Yaskawa INFORM job: DEMO_ROOF_UPPER_0625_3PAINT_61.JBI

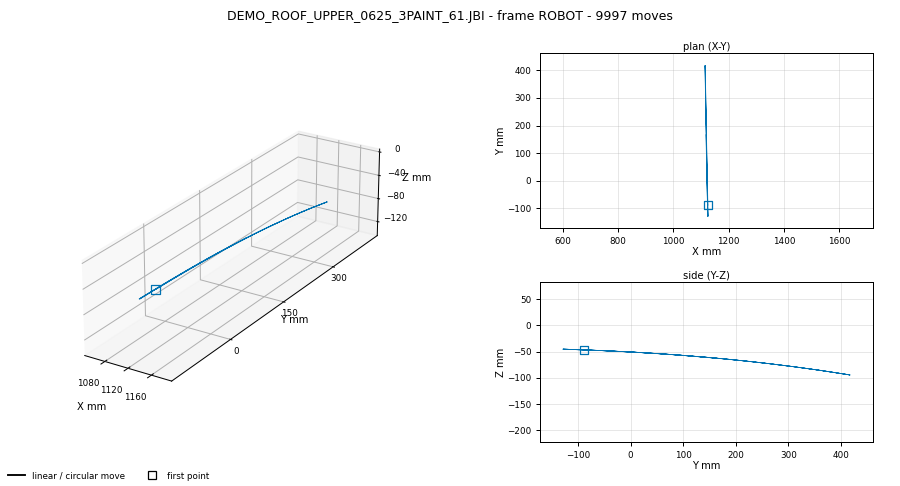
[picture p0: tool path of DEMO_ROOF_UPPER_0625_3PAINT_61.JBI in frame ROBOT, 9997 of 9997 moves have a stored position in this frame; points joined in program order, loops and branches not executed]
/JOB
//NAME DEMO_ROOF_UPPER_0625_3PAINT61
//POS
///NPOS 9997,0,0,0,0,0
///TOOL 0
///USER 0
///POSTYPE ROBOT
///RECTAN
///RCONF 1,0,0,0,0,0,0,0,0,0,0,0,0,0,0,0,0,0,0,0,0,0,0,0
C00000=1124.529,-88.514,-46.589,179.556,4.643,148.912
C00001=1124.524,-88.298,-46.597,179.556,4.647,148.913
C00002=1124.520,-88.083,-46.605,179.555,4.652,148.914
C00003=1124.516,-87.867,-46.613,179.555,4.656,148.915
C00004=1124.510,-87.651,-46.621,179.554,4.660,148.916
C00005=1124.505,-87.402,-46.630,179.554,4.665,148.917
C00006=1124.500,-87.152,-46.639,179.554,4.670,148.918
C00007=1124.494,-86.902,-46.649,179.553,4.675,148.920
C00008=1124.489,-86.652,-46.658,179.552,4.680,148.921
C00009=1124.484,-86.402,-46.667,179.552,4.685,148.922
C00010=1124.478,-86.152,-46.676,179.551,4.690,148.923
C00011=1124.473,-85.903,-46.686,179.551,4.695,148.925
C00012=1124.468,-85.653,-46.695,179.551,4.700,148.926
C00013=1124.462,-85.403,-46.704,179.551,4.705,148.927
C00014=1124.457,-85.154,-46.714,179.549,4.710,148.928
C00015=1124.452,-84.904,-46.723,179.549,4.715,148.929
C00016=1124.446,-84.654,-46.732,179.549,4.720,148.931
C00017=1124.441,-84.405,-46.742,179.549,4.725,148.932
C00018=1124.435,-84.154,-46.752,179.548,4.730,148.933
C00019=1124.430,-83.905,-46.760,179.548,4.735,148.934
C00020=1124.425,-83.655,-46.770,179.548,4.740,148.935
C00021=1124.419,-83.405,-46.780,179.548,4.745,148.936
C00022=1124.414,-83.155,-46.788,179.547,4.751,148.938
C00023=1124.409,-82.906,-46.799,179.547,4.756,148.939
C00024=1124.403,-82.656,-46.808,179.547,4.761,148.940
C00025=1124.398,-82.406,-46.817,179.546,4.766,148.941
C00026=1124.393,-82.157,-46.827,179.546,4.771,148.943
C00027=1124.388,-81.907,-46.836,179.546,4.776,148.944
C00028=1124.382,-81.657,-46.846,179.545,4.781,148.945
C00029=1124.377,-81.407,-46.855,179.545,4.786,148.946
C00030=1124.371,-81.157,-46.864,179.545,4.791,148.947
C00031=1124.366,-80.908,-46.874,179.545,4.796,148.948
C00032=1124.360,-80.658,-46.883,179.545,4.802,148.950
C00033=1124.356,-80.408,-46.893,179.545,4.807,148.951
C00034=1124.350,-80.158,-46.903,179.544,4.812,148.952
C00035=1124.345,-79.908,-46.912,179.544,4.817,148.953
C00036=1124.339,-79.658,-46.922,179.544,4.822,148.954
C00037=1124.334,-79.409,-46.931,179.544,4.827,148.955
C00038=1124.328,-79.159,-46.941,179.544,4.833,148.957
C00039=1124.324,-78.910,-46.951,179.544,4.838,148.958
C00040=1124.318,-78.659,-46.960,179.543,4.843,148.959
C00041=1124.313,-78.410,-46.970,179.543,4.848,148.960
C00042=1124.307,-78.160,-46.979,179.543,4.853,148.961
C00043=1124.302,-77.911,-46.989,179.543,4.858,148.962
C00044=1124.296,-77.661,-46.998,179.543,4.864,148.964
C00045=1124.291,-77.411,-47.008,179.543,4.870,148.965
C00046=1124.286,-77.161,-47.018,179.543,4.875,148.966
C00047=1124.280,-76.911,-47.028,179.543,4.879,148.967
C00048=1124.275,-76.662,-47.038,179.543,4.885,148.968
C00049=1124.270,-76.412,-47.047,179.543,4.890,148.969
C00050=1124.264,-76.162,-47.057,179.543,4.895,148.970
C00051=1124.259,-75.912,-47.066,179.543,4.901,148.972
C00052=1124.253,-75.663,-47.076,179.543,4.906,148.973
C00053=1124.249,-75.447,-47.084,179.543,4.910,148.974
C00054=1124.244,-75.231,-47.094,179.543,4.915,148.975
C00055=1124.240,-75.016,-47.101,179.544,4.920,148.975
C00056=1124.235,-74.800,-47.110,179.544,4.924,148.976
C00057=1124.231,-74.585,-47.118,179.544,4.928,148.977
C00058=1124.226,-74.369,-47.127,179.544,4.933,148.978
C00059=1124.222,-74.153,-47.135,179.543,4.937,148.979
C00060=1124.216,-73.938,-47.144,179.544,4.942,148.980
C00061=1124.212,-73.688,-47.153,179.544,4.947,148.981
C00062=1124.206,-73.438,-47.163,179.544,4.952,148.982
C00063=1124.201,-73.189,-47.174,179.545,4.958,148.984
C00064=1124.196,-72.939,-47.183,179.544,4.963,148.985
C00065=1124.190,-72.689,-47.193,179.545,4.968,148.986
C00066=1124.184,-72.440,-47.203,179.545,4.974,148.987
C00067=1124.179,-72.189,-47.214,179.545,4.979,148.988
C00068=1124.174,-71.940,-47.223,179.545,4.984,148.989
C00069=1124.168,-71.690,-47.233,179.546,4.990,148.990
C00070=1124.163,-71.441,-47.243,179.546,4.995,148.991
C00071=1124.158,-71.191,-47.252,179.546,5.000,148.992
C00072=1124.153,-70.941,-47.263,179.547,5.006,148.993
C00073=1124.147,-70.691,-47.273,179.547,5.010,148.994
C00074=1124.141,-70.441,-47.283,179.547,5.016,148.995
C00075=1124.137,-70.192,-47.292,179.548,5.021,148.996
C00076=1124.132,-69.942,-47.303,179.548,5.026,148.997
C00077=1124.126,-69.692,-47.313,179.549,5.032,148.998
C00078=1124.120,-69.443,-47.323,179.548,5.037,149.000
C00079=1124.116,-69.194,-47.333,179.549,5.043,149.000
C00080=1124.110,-68.943,-47.343,179.549,5.048,149.002
C00081=1124.105,-68.693,-47.353,179.550,5.053,149.003
C00082=1124.099,-68.444,-47.363,179.550,5.059,149.004
C00083=1124.094,-68.193,-47.374,179.550,5.063,149.005
C00084=1124.089,-67.944,-47.383,179.551,5.069,149.006
C00085=1124.084,-67.695,-47.394,179.551,5.074,149.007
C00086=1124.078,-67.445,-47.404,179.552,5.080,149.008
C00087=1124.073,-67.195,-47.414,179.552,5.085,149.009
C00088=1124.067,-66.945,-47.425,179.553,5.090,149.010
C00089=1124.062,-66.696,-47.435,179.554,5.095,149.011
C00090=1124.058,-66.446,-47.445,179.554,5.101,149.012
C00091=1124.052,-66.196,-47.455,179.554,5.106,149.013
C00092=1124.046,-65.947,-47.465,179.555,5.111,149.014
C00093=1124.041,-65.696,-47.476,179.555,5.117,149.015
C00094=1124.036,-65.447,-47.486,179.556,5.122,149.016
C00095=1124.030,-65.197,-47.496,179.557,5.128,149.017
C00096=1124.025,-64.947,-47.507,179.558,5.132,149.017
C00097=1124.020,-64.698,-47.517,179.559,5.138,149.018
C00098=1124.014,-64.448,-47.527,179.558,5.143,149.020
C00099=1124.010,-64.198,-47.537,179.559,5.149,149.020
C00100=1124.004,-63.949,-47.547,179.560,5.153,149.021
C00101=1123.998,-63.699,-47.558,179.561,5.159,149.022
C00102=1123.993,-63.449,-47.568,179.562,5.165,149.023
C00103=1123.988,-63.199,-47.578,179.562,5.169,149.024
C00104=1123.983,-62.950,-47.590,179.563,5.175,149.025
C00105=1123.978,-62.700,-47.600,179.564,5.180,149.026
C00106=1123.972,-62.451,-47.610,179.564,5.185,149.027
C00107=1123.967,-62.200,-47.621,179.565,5.191,149.028
C00108=1123.961,-61.951,-47.631,179.566,5.196,149.029
C00109=1123.957,-61.735,-47.640,179.567,5.201,149.030
C00110=1123.952,-61.520,-47.649,179.568,5.206,149.030
C00111=1123.948,-61.305,-47.658,179.568,5.210,149.031
C00112=1123.944,-61.089,-47.667,179.569,5.215,149.032
C00113=1123.939,-60.874,-47.677,179.570,5.219,149.033
C00114=1123.934,-60.658,-47.686,179.570,5.224,149.033
C00115=1123.929,-60.442,-47.695,179.571,5.228,149.034
C00116=1123.925,-60.226,-47.704,179.572,5.233,149.035
C00117=1123.920,-59.977,-47.715,179.571,5.237,149.036
C00118=1123.914,-59.727,-47.725,179.571,5.242,149.037
C00119=1123.909,-59.477,-47.736,179.571,5.246,149.038
C00120=1123.904,-59.228,-47.747,179.571,5.251,149.039
C00121=1123.898,-58.979,-47.757,179.571,5.256,149.040
C00122=1123.893,-58.728,-47.768,179.571,5.260,149.041
C00123=1123.888,-58.479,-47.778,179.571,5.265,149.042
C00124=1123.883,-58.229,-47.789,179.570,5.269,149.043
C00125=1123.878,-57.980,-47.799,179.570,5.274,149.045
C00126=1123.873,-57.729,-47.810,179.570,5.279,149.046
C00127=1123.867,-57.480,-47.821,179.570,5.284,149.047
C00128=1123.862,-57.230,-47.831,179.569,5.288,149.048
C00129=1123.856,-56.980,-47.842,179.569,5.293,149.049
C00130=1123.851,-56.731,-47.854,179.570,5.298,149.050
C00131=1123.846,-56.481,-47.864,179.569,5.302,149.051
C00132=1123.841,-56.232,-47.875,179.569,5.307,149.052
C00133=1123.836,-55.981,-47.886,179.569,5.311,149.053
C00134=1123.830,-55.732,-47.896,179.568,5.316,149.054
C00135=1123.826,-55.482,-47.907,179.568,5.320,149.055
C00136=1123.820,-55.233,-47.917,179.568,5.326,149.056
C00137=1123.815,-54.983,-47.929,179.568,5.331,149.057
C00138=1123.809,-54.733,-47.939,179.567,5.335,149.059
C00139=1123.804,-54.483,-47.950,179.568,5.340,149.059
C00140=1123.799,-54.234,-47.961,179.567,5.344,149.061
C00141=1123.794,-53.984,-47.972,179.567,5.349,149.062
C00142=1123.788,-53.735,-47.982,179.567,5.353,149.063
C00143=1123.783,-53.484,-47.994,179.567,5.358,149.064
C00144=1123.778,-53.235,-48.005,179.567,5.363,149.065
C00145=1123.772,-52.985,-48.015,179.567,5.367,149.066
C00146=1123.768,-52.735,-48.026,179.566,5.373,149.067
C00147=1123.762,-52.486,-48.037,179.566,5.377,149.068
C00148=1123.757,-52.236,-48.048,179.566,5.382,149.069
C00149=1123.751,-51.986,-48.059,179.565,5.386,149.070
C00150=1123.746,-51.737,-48.070,179.565,5.391,149.071
C00151=1123.741,-51.487,-48.081,179.566,5.396,149.072
C00152=1123.735,-51.237,-48.092,179.565,5.400,149.073
C00153=1123.730,-50.987,-48.103,179.565,5.405,149.075
C00154=1123.725,-50.738,-48.114,179.565,5.409,149.075
C00155=1123.720,-50.488,-48.124,179.565,5.415,149.077
C00156=1123.714,-50.239,-48.136,179.564,5.419,149.078
C00157=1123.709,-49.988,-48.146,179.564,5.424,149.079
C00158=1123.704,-49.739,-48.158,179.564,5.429,149.080
C00159=1123.698,-49.490,-48.169,179.564,5.433,149.081
C00160=1123.693,-49.239,-48.180,179.564,5.438,149.082
C00161=1123.689,-48.990,-48.191,179.564,5.442,149.083
C00162=1123.683,-48.740,-48.201,179.563,5.447,149.084
C00163=1123.678,-48.490,-48.213,179.563,5.452,149.085
C00164=1123.672,-48.241,-48.224,179.563,5.457,149.086
C00165=1123.668,-48.026,-48.233,179.563,5.461,149.087
C00166=1123.664,-47.810,-48.243,179.562,5.465,149.088
C00167=1123.659,-47.594,-48.252,179.562,5.469,149.089
C00168=1123.655,-47.379,-48.262,179.562,5.473,149.090
C00169=1123.650,-47.164,-48.271,179.562,5.477,149.091
C00170=1123.645,-46.948,-48.281,179.562,5.481,149.092
C00171=1123.641,-46.733,-48.291,179.562,5.485,149.093
C00172=1123.636,-46.518,-48.300,179.562,5.489,149.094
C00173=1123.631,-46.268,-48.312,179.561,5.494,149.095
C00174=1123.625,-46.018,-48.322,179.561,5.499,149.096
C00175=1123.620,-45.768,-48.334,179.562,5.503,149.097
C00176=1123.615,-45.519,-48.345,179.561,5.508,149.098
C00177=1123.610,-45.269,-48.356,179.561,5.513,149.099
C00178=1123.604,-45.019,-48.367,179.560,5.517,149.100
C00179=1123.600,-44.770,-48.379,179.561,5.522,149.101
C00180=1123.595,-44.520,-48.390,179.561,5.527,149.102
C00181=1123.589,-44.270,-48.401,179.560,5.532,149.104
C00182=1123.584,-44.021,-48.412,179.560,5.536,149.105
C00183=1123.578,-43.771,-48.424,179.560,5.541,149.106
C00184=1123.573,-43.521,-48.434,179.560,5.546,149.107
C00185=1123.568,-43.272,-48.445,179.559,5.550,149.108
C00186=1123.563,-43.022,-48.457,179.560,5.556,149.109
C00187=1123.557,-42.773,-48.468,179.562,5.561,149.109
C00188=1123.552,-42.523,-48.480,179.563,5.567,149.110
C00189=1123.547,-42.273,-48.491,179.565,5.572,149.111
C00190=1123.542,-42.023,-48.503,179.567,5.578,149.112
C00191=1123.536,-41.774,-48.514,179.568,5.584,149.113
C00192=1123.531,-41.524,-48.525,179.570,5.590,149.113
C00193=1123.526,-41.274,-48.537,179.572,5.595,149.114
C00194=1123.521,-41.024,-48.549,179.573,5.600,149.115
C00195=1123.515,-40.775,-48.560,179.574,5.606,149.115
C00196=1123.510,-40.525,-48.571,179.576,5.611,149.116
C00197=1123.505,-40.275,-48.582,179.577,5.617,149.117
C00198=1123.500,-40.025,-48.594,179.579,5.622,149.118
C00199=1123.494,-39.776,-48.605,179.580,5.627,149.118
C00200=1123.489,-39.526,-48.617,179.581,5.632,149.119
C00201=1123.484,-39.277,-48.628,179.582,5.637,149.120
C00202=1123.479,-39.027,-48.640,179.583,5.643,149.121
C00203=1123.473,-38.777,-48.652,179.585,5.648,149.122
C00204=1123.468,-38.528,-48.663,179.586,5.653,149.122
C00205=1123.463,-38.278,-48.675,179.587,5.658,149.123
C00206=1123.458,-38.028,-48.686,179.588,5.663,149.124
C00207=1123.452,-37.778,-48.698,179.589,5.668,149.125
C00208=1123.447,-37.528,-48.710,179.590,5.673,149.125
C00209=1123.442,-37.279,-48.721,179.591,5.678,149.126
C00210=1123.437,-37.029,-48.734,179.592,5.683,149.127
C00211=1123.432,-36.781,-48.744,179.593,5.688,149.128
C00212=1123.426,-36.531,-48.756,179.594,5.693,149.128
C00213=1123.421,-36.281,-48.768,179.595,5.698,149.129
C00214=1123.416,-36.031,-48.779,179.595,5.702,149.130
C00215=1123.411,-35.781,-48.791,179.596,5.707,149.131
C00216=1123.405,-35.531,-48.803,179.597,5.711,149.132
C00217=1123.400,-35.281,-48.815,179.598,5.716,149.133
C00218=1123.396,-35.032,-48.827,179.598,5.721,149.133
C00219=1123.390,-34.783,-48.839,179.598,5.725,149.134
C00220=1123.384,-34.533,-48.851,179.599,5.730,149.135
C00221=1123.380,-34.317,-48.861,179.600,5.734,149.136
C00222=1123.376,-34.103,-48.871,179.600,5.738,149.137
C00223=1123.371,-33.887,-48.881,179.601,5.741,149.137
C00224=1123.367,-33.671,-48.891,179.601,5.746,149.138
C00225=1123.362,-33.456,-48.902,179.601,5.750,149.139
C00226=1123.358,-33.241,-48.912,179.602,5.753,149.139
C00227=1123.353,-33.026,-48.922,179.602,5.757,149.140
C00228=1123.349,-32.810,-48.933,179.602,5.761,149.141
C00229=1123.344,-32.561,-48.944,179.602,5.766,149.142
C00230=1123.339,-32.311,-48.956,179.602,5.770,149.143
C00231=1123.333,-32.061,-48.968,179.603,5.774,149.144
C00232=1123.328,-31.812,-48.980,179.603,5.778,149.145
C00233=1123.322,-31.562,-48.992,179.603,5.783,149.146
C00234=1123.317,-31.313,-49.003,179.603,5.787,149.146
C00235=1123.312,-31.063,-49.015,179.603,5.791,149.147
C00236=1123.307,-30.813,-49.028,179.603,5.796,149.148
C00237=1123.301,-30.564,-49.040,179.603,5.800,149.149
C00238=1123.297,-30.314,-49.051,179.602,5.804,149.150
C00239=1123.292,-30.065,-49.064,179.602,5.808,149.151
C00240=1123.286,-29.815,-49.075,179.602,5.812,149.152
C00241=1123.281,-29.565,-49.087,179.602,5.817,149.153
C00242=1123.276,-29.315,-49.100,179.602,5.821,149.154
C00243=1123.270,-29.065,-49.112,179.601,5.825,149.155
C00244=1123.265,-28.816,-49.123,179.601,5.829,149.156
C00245=1123.260,-28.567,-49.136,179.600,5.833,149.157
C00246=1123.255,-28.317,-49.148,179.599,5.837,149.158
C00247=1123.250,-28.067,-49.160,179.599,5.841,149.159
C00248=1123.244,-27.817,-49.172,179.599,5.845,149.161
C00249=1123.239,-27.567,-49.184,179.598,5.850,149.162
C00250=1123.235,-27.318,-49.196,179.598,5.854,149.163
C00251=1123.229,-27.068,-49.208,179.597,5.857,149.164
C00252=1123.224,-26.819,-49.220,179.596,5.861,149.165
C00253=1123.219,-26.569,-49.232,179.595,5.866,149.166
C00254=1123.213,-26.319,-49.244,179.594,5.869,149.167
C00255=1123.208,-26.070,-49.257,179.594,5.874,149.168
C00256=1123.203,-25.820,-49.269,179.593,5.878,149.169
C00257=1123.198,-25.571,-49.281,179.593,5.883,149.170
C00258=1123.193,-25.321,-49.293,179.595,5.888,149.171
C00259=1123.188,-25.072,-49.305,179.595,5.893,149.172
C00260=1123.182,-24.822,-49.317,179.596,5.897,149.173
C00261=1123.177,-24.571,-49.329,179.597,5.903,149.174
C00262=1123.172,-24.322,-49.342,179.597,5.908,149.174
C00263=1123.167,-24.072,-49.354,179.598,5.912,149.175
C00264=1123.162,-23.823,-49.366,179.598,5.917,149.176
C00265=1123.156,-23.573,-49.378,179.599,5.923,149.177
C00266=1123.151,-23.323,-49.391,179.600,5.927,149.178
C00267=1123.146,-23.073,-49.403,179.601,5.932,149.179
C00268=1123.141,-22.824,-49.415,179.601,5.936,149.180
C00269=1123.135,-22.575,-49.428,179.602,5.942,149.181
C00270=1123.130,-22.325,-49.440,179.603,5.947,149.181
C00271=1123.125,-22.076,-49.452,179.603,5.951,149.182
C00272=1123.119,-21.826,-49.464,179.604,5.956,149.183
C00273=1123.114,-21.576,-49.477,179.605,5.961,149.184
C00274=1123.109,-21.326,-49.489,179.606,5.966,149.185
C00275=1123.104,-21.076,-49.502,179.606,5.971,149.186
C00276=1123.099,-20.827,-49.514,179.607,5.975,149.187
C00277=1123.095,-20.612,-49.524,179.608,5.980,149.187
C00278=1123.090,-20.396,-49.535,179.608,5.983,149.188
C00279=1123.085,-20.181,-49.546,179.609,5.988,149.189
C00280=1123.081,-19.967,-49.557,179.610,5.992,149.189
C00281=1123.077,-19.751,-49.568,179.610,5.996,149.190
C00282=1123.073,-19.536,-49.578,179.611,6.000,149.191
C00283=1123.068,-19.320,-49.589,179.611,6.004,149.191
C00284=1123.063,-19.106,-49.600,179.612,6.009,149.192
C00285=1123.058,-18.856,-49.612,179.613,6.013,149.193
C00286=1123.053,-18.606,-49.624,179.613,6.018,149.194
C00287=1123.048,-18.356,-49.637,179.614,6.022,149.195
C00288=1123.043,-18.106,-49.649,179.614,6.027,149.196
C00289=1123.038,-17.857,-49.662,179.616,6.032,149.196
C00290=1123.033,-17.608,-49.674,179.616,6.037,149.197
C00291=1123.027,-17.358,-49.687,179.617,6.042,149.198
C00292=1123.022,-17.108,-49.701,179.617,6.047,149.199
C00293=1123.017,-16.858,-49.712,179.618,6.051,149.200
C00294=1123.012,-16.609,-49.725,179.619,6.056,149.201
C00295=1123.006,-16.360,-49.738,179.619,6.060,149.201
C00296=1123.001,-16.110,-49.750,179.620,6.065,149.202
C00297=1122.997,-15.860,-49.763,179.621,6.069,149.203
C00298=1122.991,-15.610,-49.776,179.621,6.074,149.204
C00299=1122.986,-15.361,-49.788,179.622,6.079,149.205
C00300=1122.980,-15.111,-49.801,179.623,6.084,149.205
C00301=1122.975,-14.862,-49.814,179.624,6.089,149.206
C00302=1122.971,-14.612,-49.827,179.624,6.093,149.207
C00303=1122.966,-14.363,-49.839,179.625,6.098,149.208
C00304=1122.960,-14.113,-49.852,179.626,6.103,149.209
C00305=1122.954,-13.863,-49.864,179.626,6.107,149.210
C00306=1122.950,-13.613,-49.877,179.627,6.112,149.210
C00307=1122.945,-13.364,-49.890,179.628,6.116,149.211
C00308=1122.939,-13.114,-49.903,179.628,6.121,149.212
C00309=1122.934,-12.864,-49.916,179.629,6.126,149.213
C00310=1122.929,-12.615,-49.929,179.630,6.130,149.214
C00311=1122.924,-12.365,-49.941,179.630,6.135,149.215
C00312=1122.918,-12.116,-49.954,179.631,6.140,149.215
C00313=1122.914,-11.866,-49.967,179.632,6.144,149.216
C00314=1122.909,-11.617,-49.980,179.632,6.149,149.217
C00315=1122.903,-11.367,-49.992,179.633,6.153,149.218
C00316=1122.898,-11.117,-50.006,179.634,6.158,149.219
C00317=1122.893,-10.868,-50.019,179.634,6.162,149.219
C00318=1122.888,-10.618,-50.031,179.635,6.167,149.220
C00319=1122.882,-10.369,-50.044,179.636,6.172,149.221
C00320=1122.878,-10.119,-50.057,179.636,6.176,149.222
C00321=1122.872,-9.869,-50.070,179.637,6.181,149.223
C00322=1122.867,-9.620,-50.083,179.638,6.185,149.223
C00323=1122.862,-9.370,-50.096,179.638,6.190,149.224
C00324=1122.857,-9.121,-50.109,179.639,6.195,149.225
C00325=1122.853,-8.871,-50.122,179.640,6.199,149.226
C00326=1122.847,-8.621,-50.136,179.640,6.204,149.227
C00327=1122.842,-8.372,-50.148,179.641,6.209,149.228
C00328=1122.836,-8.122,-50.162,179.642,6.213,149.228
C00329=1122.831,-7.872,-50.174,179.642,6.218,149.229
C00330=1122.826,-7.623,-50.187,179.643,6.222,149.230
C00331=1122.821,-7.373,-50.201,179.644,6.227,149.231
C00332=1122.816,-7.124,-50.214,179.644,6.231,149.232
C00333=1122.812,-6.908,-50.225,179.645,6.235,149.232
C00334=1122.807,-6.694,-50.236,179.645,6.239,149.233
C00335=1122.803,-6.478,-50.248,179.646,6.243,149.234
C00336=1122.799,-6.263,-50.260,179.646,6.247,149.234
C00337=1122.793,-6.048,-50.270,179.646,6.250,149.235
C00338=1122.789,-5.833,-50.282,179.647,6.255,149.236
C00339=1122.785,-5.618,-50.293,179.648,6.258,149.236
C00340=1122.780,-5.403,-50.305,179.649,6.263,149.237
C00341=1122.775,-5.153,-50.317,179.649,6.267,149.238
C00342=1122.770,-4.903,-50.331,179.649,6.271,149.239
C00343=1122.765,-4.654,-50.344,179.650,6.276,149.240
C00344=1122.760,-4.404,-50.358,179.651,6.280,149.240
C00345=1122.755,-4.155,-50.370,179.651,6.285,149.241
C00346=1122.750,-3.905,-50.383,179.652,6.290,149.242
C00347=1122.744,-3.655,-50.397,179.653,6.294,149.243
C00348=1122.740,-3.406,-50.410,179.653,6.299,149.244
C00349=1122.734,-3.156,-50.424,179.654,6.304,149.245
C00350=1122.729,-2.907,-50.436,179.655,6.308,149.245
C00351=1122.724,-2.657,-50.450,179.655,6.312,149.246
C00352=1122.718,-2.407,-50.464,179.655,6.317,149.247
C00353=1122.714,-2.157,-50.477,179.656,6.321,149.248
C00354=1122.708,-1.908,-50.490,179.657,6.326,149.249
C00355=1122.704,-1.658,-50.503,179.657,6.330,149.250
C00356=1122.698,-1.409,-50.517,179.658,6.335,149.250
C00357=1122.694,-1.159,-50.530,179.659,6.339,149.251
C00358=1122.688,-0.910,-50.544,179.659,6.343,149.252
C00359=1122.684,-0.660,-50.557,179.659,6.348,149.253
C00360=1122.678,-0.411,-50.570,179.660,6.353,149.254
C00361=1122.673,-0.161,-50.585,179.661,6.357,149.254
C00362=1122.668,0.088,-50.597,179.661,6.362,149.255
C00363=1122.662,0.339,-50.611,179.662,6.367,149.256
C00364=1122.658,0.587,-50.624,179.662,6.371,149.257
C00365=1122.652,0.838,-50.638,179.663,6.375,149.258
C00366=1122.647,1.087,-50.652,179.663,6.379,149.259
C00367=1122.642,1.337,-50.665,179.664,6.384,149.259
C00368=1122.637,1.586,-50.678,179.664,6.389,149.260
C00369=1122.632,1.836,-50.691,179.665,6.393,149.261
C00370=1122.627,2.085,-50.705,179.666,6.398,149.262
C00371=1122.621,2.335,-50.719,179.666,6.403,149.263
C00372=1122.617,2.584,-50.732,179.666,6.407,149.264
C00373=1122.611,2.834,-50.746,179.667,6.411,149.265
C00374=1122.606,3.083,-50.760,179.668,6.416,149.265
C00375=1122.601,3.333,-50.773,179.668,6.420,149.266
C00376=1122.596,3.583,-50.787,179.669,6.425,149.267
C00377=1122.591,3.832,-50.801,179.669,6.429,149.268
C00378=1122.586,4.082,-50.814,179.669,6.434,149.269
C00379=1122.581,4.331,-50.828,179.670,6.438,149.269
C00380=1122.575,4.581,-50.841,179.671,6.443,149.270
C00381=1122.570,4.831,-50.856,179.672,6.448,149.271
C00382=1122.566,5.080,-50.869,179.672,6.452,149.272
C00383=1122.560,5.330,-50.882,179.672,6.456,149.273
C00384=1122.555,5.579,-50.896,179.673,6.461,149.274
C00385=1122.550,5.829,-50.911,179.673,6.466,149.275
C00386=1122.545,6.079,-50.924,179.674,6.470,149.275
C00387=1122.540,6.328,-50.938,179.675,6.475,149.276
C00388=1122.535,6.577,-50.952,179.675,6.479,149.277
C00389=1122.531,6.793,-50.963,179.675,6.483,149.278
C00390=1122.526,7.007,-50.975,179.676,6.487,149.279
C00391=1122.522,7.223,-50.986,179.676,6.490,149.279
C00392=1122.517,7.438,-50.999,179.676,6.495,149.280
C00393=1122.513,7.653,-51.011,179.677,6.499,149.281
C00394=1122.508,7.867,-51.022,179.677,6.502,149.282
C00395=1122.504,8.083,-51.034,179.677,6.506,149.282
C00396=1122.499,8.298,-51.046,179.678,6.510,149.283
C00397=1122.495,8.548,-51.060,179.679,6.515,149.284
C00398=1122.489,8.797,-51.074,179.679,6.520,149.285
C00399=1122.484,9.046,-51.088,179.680,6.524,149.285
C00400=1122.479,9.297,-51.102,179.681,6.529,149.286
C00401=1122.473,9.546,-51.116,179.681,6.534,149.287
C00402=1122.469,9.795,-51.130,179.682,6.538,149.288
C00403=1122.464,10.045,-51.144,179.683,6.543,149.289
C00404=1122.459,10.294,-51.158,179.684,6.548,149.290
C00405=1122.453,10.544,-51.171,179.685,6.552,149.290
C00406=1122.449,10.794,-51.185,179.686,6.557,149.291
C00407=1122.443,11.043,-51.199,179.686,6.562,149.292
C00408=1122.438,11.292,-51.214,179.687,6.566,149.293
C00409=1122.433,11.542,-51.228,179.688,6.571,149.294
C00410=1122.428,11.792,-51.242,179.689,6.575,149.294
C00411=1122.423,12.041,-51.256,179.689,6.580,149.295
C00412=1122.418,12.290,-51.270,179.690,6.585,149.296
C00413=1122.413,12.541,-51.283,179.691,6.589,149.297
C00414=1122.408,12.790,-51.298,179.692,6.594,149.298
C00415=1122.403,13.039,-51.312,179.693,6.599,149.298
C00416=1122.398,13.289,-51.326,179.694,6.604,149.299
C00417=1122.393,13.539,-51.340,179.695,6.608,149.300
C00418=1122.388,13.788,-51.354,179.695,6.613,149.301
C00419=1122.382,14.037,-51.368,179.696,6.617,149.301
C00420=1122.377,14.287,-51.383,179.697,6.622,149.302
C00421=1122.372,14.537,-51.397,179.698,6.626,149.303
C00422=1122.367,14.787,-51.411,179.699,6.631,149.304
C00423=1122.362,15.036,-51.425,179.699,6.635,149.305
C00424=1122.357,15.285,-51.439,179.700,6.640,149.305
C00425=1122.352,15.535,-51.454,179.701,6.644,149.306
C00426=1122.347,15.785,-51.468,179.702,6.649,149.307
C00427=1122.342,16.034,-51.482,179.703,6.653,149.307
C00428=1122.336,16.283,-51.496,179.703,6.658,149.308
C00429=1122.331,16.533,-51.510,179.705,6.663,149.309
C00430=1122.326,16.783,-51.525,179.706,6.668,149.310
C00431=1122.322,17.032,-51.540,179.707,6.672,149.310
C00432=1122.317,17.282,-51.554,179.707,6.677,149.311
C00433=1122.311,17.531,-51.568,179.708,6.681,149.312
C00434=1122.306,17.780,-51.582,179.709,6.685,149.313
C00435=1122.301,18.030,-51.596,179.710,6.690,149.313
C00436=1122.296,18.280,-51.611,179.711,6.694,149.314
C00437=1122.291,18.530,-51.626,179.711,6.699,149.315
C00438=1122.286,18.779,-51.641,179.712,6.703,149.316
C00439=1122.281,19.028,-51.654,179.713,6.708,149.316
C00440=1122.276,19.278,-51.669,179.714,6.712,149.317
C00441=1122.271,19.527,-51.683,179.715,6.717,149.318
C00442=1122.266,19.777,-51.697,179.716,6.721,149.318
C00443=1122.261,20.026,-51.712,179.717,6.726,149.319
C00444=1122.256,20.276,-51.727,179.718,6.730,149.320
C00445=1122.251,20.491,-51.739,179.719,6.734,149.321
C00446=1122.247,20.706,-51.752,179.719,6.738,149.321
C00447=1122.243,20.921,-51.764,179.720,6.742,149.322
C00448=1122.238,21.136,-51.777,179.721,6.745,149.322
C00449=1122.234,21.351,-51.789,179.722,6.750,149.323
C00450=1122.229,21.566,-51.802,179.723,6.753,149.324
C00451=1122.225,21.781,-51.814,179.724,6.758,149.324
C00452=1122.221,21.996,-51.827,179.724,6.761,149.325
C00453=1122.215,22.245,-51.841,179.725,6.765,149.326
C00454=1122.210,22.495,-51.855,179.726,6.770,149.326
C00455=1122.206,22.744,-51.870,179.727,6.774,149.327
C00456=1122.200,22.994,-51.885,179.728,6.779,149.328
C00457=1122.195,23.243,-51.900,179.729,6.783,149.328
C00458=1122.190,23.492,-51.915,179.730,6.787,149.329
C00459=1122.185,23.742,-51.929,179.731,6.792,149.330
C00460=1122.180,23.992,-51.944,179.732,6.796,149.331
C00461=1122.175,24.241,-51.959,179.733,6.801,149.331
C00462=1122.170,24.491,-51.973,179.734,6.805,149.332
C00463=1122.165,24.740,-51.988,179.735,6.809,149.333
C00464=1122.160,24.990,-52.003,179.736,6.814,149.333
C00465=1122.155,25.240,-52.017,179.737,6.818,149.334
C00466=1122.150,25.489,-52.032,179.737,6.823,149.335
C00467=1122.144,25.739,-52.047,179.738,6.827,149.335
C00468=1122.140,25.988,-52.062,179.739,6.831,149.336
C00469=1122.135,26.238,-52.076,179.741,6.836,149.337
C00470=1122.130,26.487,-52.092,179.742,6.840,149.337
C00471=1122.125,26.737,-52.106,179.743,6.844,149.338
C00472=1122.120,26.986,-52.121,179.744,6.849,149.339
C00473=1122.114,27.236,-52.136,179.744,6.853,149.340
C00474=1122.110,27.485,-52.151,179.745,6.858,149.340
C00475=1122.105,27.735,-52.165,179.746,6.862,149.341
C00476=1122.099,27.984,-52.181,179.747,6.866,149.342
C00477=1122.094,28.234,-52.195,179.748,6.871,149.342
C00478=1122.090,28.483,-52.210,179.750,6.875,149.343
C00479=1122.084,28.732,-52.226,179.751,6.879,149.343
C00480=1122.079,28.982,-52.240,179.752,6.883,149.344
C00481=1122.074,29.231,-52.256,179.753,6.888,149.345
C00482=1122.069,29.481,-52.270,179.754,6.892,149.345
C00483=1122.064,29.730,-52.285,179.755,6.896,149.346
C00484=1122.059,29.980,-52.300,179.756,6.901,149.347
C00485=1122.054,30.229,-52.315,179.757,6.905,149.347
C00486=1122.049,30.479,-52.330,179.758,6.909,149.348
C00487=1122.044,30.728,-52.345,179.759,6.914,149.349
C00488=1122.039,30.979,-52.361,179.760,6.918,149.349
C00489=1122.034,31.228,-52.376,179.761,6.922,149.350
C00490=1122.030,31.477,-52.391,179.762,6.927,149.351
C00491=1122.024,31.727,-52.405,179.763,6.931,149.351
C00492=1122.019,31.976,-52.420,179.764,6.935,149.352
C00493=1122.014,32.225,-52.436,179.765,6.940,149.353
C00494=1122.009,32.475,-52.450,179.766,6.944,149.353
C00495=1122.003,32.724,-52.466,179.768,6.948,149.354
C00496=1121.999,32.974,-52.481,179.769,6.952,149.355
C00497=1121.994,33.224,-52.497,179.770,6.957,149.355
C00498=1121.989,33.473,-52.511,179.771,6.961,149.356
C00499=1121.984,33.723,-52.527,179.772,6.965,149.356
C00500=1121.978,33.972,-52.542,179.772,6.969,149.357
C00501=1121.974,34.187,-52.555,179.774,6.973,149.358
C00502=1121.970,34.401,-52.568,179.774,6.976,149.358
C00503=1121.966,34.616,-52.581,179.776,6.980,149.359
C00504=1121.962,34.832,-52.595,179.776,6.984,149.359
C00505=1121.957,35.047,-52.608,179.778,6.988,149.360
C00506=1121.953,35.261,-52.621,179.778,6.991,149.360
C00507=1121.948,35.476,-52.634,179.779,6.994,149.361
C00508=1121.944,35.691,-52.647,179.780,6.999,149.361
C00509=1121.939,35.940,-52.662,179.781,7.003,149.362
C00510=1121.934,36.190,-52.678,179.782,7.007,149.363
C00511=1121.929,36.439,-52.693,179.783,7.012,149.363
C00512=1121.924,36.689,-52.709,179.785,7.016,149.364
C00513=1121.919,36.938,-52.724,179.786,7.020,149.364
C00514=1121.914,37.187,-52.739,179.786,7.023,149.365
C00515=1121.908,37.437,-52.754,179.787,7.028,149.366
C00516=1121.904,37.687,-52.770,179.789,7.032,149.366
C00517=1121.899,37.936,-52.785,179.790,7.036,149.367
C00518=1121.893,38.186,-52.801,179.791,7.040,149.368
C00519=1121.889,38.435,-52.816,179.792,7.045,149.368
C00520=1121.884,38.685,-52.832,179.793,7.049,149.369
C00521=1121.879,38.934,-52.847,179.794,7.053,149.369
C00522=1121.873,39.184,-52.863,179.795,7.057,149.370
C00523=1121.869,39.433,-52.878,179.797,7.061,149.371
C00524=1121.864,39.683,-52.894,179.798,7.066,149.371
C00525=1121.858,39.932,-52.910,179.799,7.070,149.372
C00526=1121.854,40.181,-52.925,179.800,7.074,149.372
C00527=1121.849,40.430,-52.941,179.801,7.079,149.373
C00528=1121.844,40.680,-52.957,179.803,7.083,149.374
C00529=1121.838,40.930,-52.972,179.804,7.087,149.374
C00530=1121.834,41.179,-52.987,179.805,7.091,149.375
C00531=1121.828,41.428,-53.003,179.806,7.095,149.375
C00532=1121.824,41.678,-53.019,179.807,7.099,149.376
C00533=1121.818,41.928,-53.035,179.808,7.103,149.377
C00534=1121.814,42.177,-53.050,179.809,7.107,149.377
C00535=1121.809,42.427,-53.065,179.810,7.112,149.378
C00536=1121.804,42.676,-53.082,179.812,7.115,149.378
C00537=1121.798,42.925,-53.097,179.813,7.120,149.379
C00538=1121.794,43.175,-53.113,179.814,7.124,149.380
C00539=1121.789,43.424,-53.128,179.815,7.128,149.380
C00540=1121.784,43.674,-53.144,179.817,7.132,149.381
C00541=1121.779,43.923,-53.161,179.818,7.137,149.381
C00542=1121.774,44.173,-53.176,179.819,7.141,149.382
C00543=1121.768,44.422,-53.192,179.820,7.145,149.382
C00544=1121.763,44.672,-53.208,179.821,7.149,149.383
C00545=1121.759,44.921,-53.223,179.822,7.153,149.384
C00546=1121.754,45.170,-53.239,179.824,7.157,149.384
C00547=1121.749,45.420,-53.255,179.824,7.161,149.385
C00548=1121.744,45.669,-53.271,179.825,7.165,149.385
C00549=1121.739,45.918,-53.287,179.827,7.169,149.386
C00550=1121.734,46.168,-53.303,179.828,7.173,149.386
C00551=1121.728,46.418,-53.318,179.830,7.177,149.387
C00552=1121.724,46.667,-53.335,179.831,7.182,149.388
C00553=1121.719,46.916,-53.350,179.832,7.186,149.388
C00554=1121.714,47.166,-53.366,179.833,7.190,149.389
C00555=1121.709,47.415,-53.382,179.834,7.194,149.389
C00556=1121.704,47.665,-53.398,179.836,7.198,149.390
C00557=1121.700,47.880,-53.412,179.836,7.202,149.390
C00558=1121.695,48.095,-53.426,179.838,7.205,149.391
C00559=1121.691,48.309,-53.439,179.839,7.209,149.391
C00560=1121.687,48.524,-53.453,179.839,7.212,149.392
C00561=1121.683,48.739,-53.467,179.841,7.216,149.392
C00562=1121.678,48.953,-53.481,179.842,7.219,149.393
C00563=1121.674,49.169,-53.494,179.843,7.223,149.393
C00564=1121.669,49.383,-53.508,179.844,7.227,149.394
C00565=1121.664,49.632,-53.525,179.845,7.231,149.394
C00566=1121.659,49.882,-53.541,179.847,7.235,149.395
C00567=1121.654,50.131,-53.557,179.848,7.239,149.395
C00568=1121.650,50.381,-53.573,179.849,7.243,149.396
C00569=1121.644,50.630,-53.589,179.851,7.247,149.396
C00570=1121.640,50.880,-53.605,179.851,7.250,149.397
C00571=1121.635,51.129,-53.621,179.853,7.254,149.397
C00572=1121.630,51.379,-53.637,179.854,7.259,149.398
C00573=1121.625,51.628,-53.654,179.855,7.263,149.399
C00574=1121.620,51.878,-53.670,179.856,7.267,149.399
C00575=1121.615,52.126,-53.686,179.858,7.271,149.400
C00576=1121.610,52.377,-53.702,179.859,7.275,149.400
C00577=1121.605,52.625,-53.718,179.860,7.279,149.401
C00578=1121.601,52.875,-53.735,179.862,7.283,149.401
C00579=1121.595,53.124,-53.750,179.863,7.288,149.402
C00580=1121.591,53.374,-53.767,179.864,7.292,149.402
C00581=1121.585,53.623,-53.783,179.865,7.296,149.403
C00582=1121.580,53.873,-53.800,179.867,7.300,149.404
C00583=1121.575,54.122,-53.816,179.868,7.303,149.404
C00584=1121.570,54.372,-53.832,179.869,7.307,149.405
C00585=1121.565,54.621,-53.849,179.870,7.311,149.405
C00586=1121.561,54.870,-53.865,179.872,7.315,149.406
C00587=1121.555,55.119,-53.881,179.873,7.320,149.406
C00588=1121.550,55.369,-53.898,179.874,7.324,149.407
C00589=1121.546,55.619,-53.915,179.875,7.328,149.407
C00590=1121.540,55.868,-53.930,179.877,7.332,149.408
C00591=1121.536,56.118,-53.947,179.878,7.336,149.408
C00592=1121.531,56.366,-53.963,179.880,7.340,149.409
C00593=1121.526,56.616,-53.980,179.881,7.344,149.410
C00594=1121.520,56.866,-53.996,179.882,7.348,149.410
C00595=1121.516,57.115,-54.013,179.883,7.351,149.410
C00596=1121.511,57.365,-54.030,179.884,7.356,149.411
C00597=1121.506,57.613,-54.046,179.886,7.360,149.411
C00598=1121.501,57.863,-54.063,179.887,7.364,149.412
C00599=1121.495,58.113,-54.079,179.889,7.368,149.413
C00600=1121.491,58.362,-54.095,179.890,7.372,149.413
C00601=1121.486,58.612,-54.112,179.891,7.376,149.414
C00602=1121.481,58.861,-54.129,179.892,7.380,149.414
C00603=1121.476,59.110,-54.146,179.894,7.384,149.415
C00604=1121.472,59.360,-54.162,179.895,7.388,149.415
C00605=1121.466,59.609,-54.178,179.897,7.392,149.416
C00606=1121.461,59.859,-54.195,179.898,7.396,149.416
C00607=1121.457,60.108,-54.212,179.899,7.401,149.417
C00608=1121.451,60.357,-54.228,179.900,7.404,149.417
C00609=1121.446,60.607,-54.245,179.902,7.408,149.418
C00610=1121.442,60.856,-54.262,179.903,7.412,149.418
C00611=1121.437,61.105,-54.278,179.904,7.416,149.419
C00612=1121.431,61.355,-54.296,179.906,7.420,149.419
C00613=1121.427,61.569,-54.309,179.907,7.424,149.420
C00614=1121.423,61.785,-54.324,179.908,7.427,149.420
C00615=1121.419,61.998,-54.338,179.909,7.430,149.421
C00616=1121.414,62.214,-54.353,179.911,7.434,149.421
C00617=1121.411,62.429,-54.367,179.911,7.437,149.422
C00618=1121.406,62.643,-54.382,179.912,7.440,149.422
C00619=1121.402,62.858,-54.396,179.914,7.444,149.422
C00620=1121.397,63.072,-54.411,179.915,7.447,149.423
C00621=1121.393,63.321,-54.428,179.916,7.451,149.423
C00622=1121.388,63.571,-54.445,179.918,7.456,149.424
C00623=1121.383,63.820,-54.461,179.919,7.460,149.424
C00624=1121.378,64.069,-54.478,179.921,7.463,149.425
C00625=1121.373,64.319,-54.495,179.922,7.468,149.425
C00626=1121.368,64.569,-54.512,179.923,7.472,149.426
C00627=1121.363,64.818,-54.529,179.925,7.476,149.426
C00628=1121.358,65.067,-54.546,179.926,7.480,149.427
C00629=1121.353,65.317,-54.563,179.928,7.484,149.427
C00630=1121.348,65.566,-54.580,179.928,7.487,149.428
C00631=1121.343,65.815,-54.596,179.930,7.491,149.428
C00632=1121.339,66.064,-54.614,179.931,7.495,149.429
C00633=1121.334,66.314,-54.631,179.932,7.499,149.430
C00634=1121.329,66.564,-54.648,179.934,7.503,149.430
C00635=1121.324,66.813,-54.664,179.936,7.507,149.430
C00636=1121.319,67.062,-54.681,179.937,7.511,149.431
C00637=1121.314,67.311,-54.699,179.938,7.515,149.431
C00638=1121.309,67.561,-54.716,179.940,7.519,149.432
C00639=1121.305,67.810,-54.733,179.941,7.523,149.432
C00640=1121.299,68.060,-54.750,179.942,7.527,149.433
C00641=1121.294,68.309,-54.768,179.944,7.531,149.433
C00642=1121.289,68.558,-54.784,179.946,7.535,149.434
C00643=1121.284,68.808,-54.801,179.947,7.540,149.434
C00644=1121.280,69.057,-54.818,179.948,7.543,149.435
C00645=1121.275,69.307,-54.836,179.949,7.547,149.435
C00646=1121.270,69.555,-54.852,179.950,7.551,149.436
C00647=1121.265,69.805,-54.870,179.952,7.555,149.436
C00648=1121.260,70.054,-54.888,179.953,7.559,149.437
C00649=1121.255,70.304,-54.904,179.955,7.563,149.437
C00650=1121.250,70.554,-54.922,179.956,7.567,149.438
C00651=1121.246,70.802,-54.939,179.958,7.571,149.438
C00652=1121.241,71.052,-54.956,179.959,7.575,149.439
C00653=1121.235,71.301,-54.973,179.960,7.579,149.439
C00654=1121.231,71.550,-54.991,179.962,7.583,149.440
C00655=1121.225,71.800,-55.008,179.964,7.587,149.440
C00656=1121.220,72.049,-55.026,179.965,7.591,149.441
C00657=1121.216,72.299,-55.042,179.966,7.595,149.441
C00658=1121.211,72.548,-55.060,179.968,7.599,149.442
C00659=1121.206,72.798,-55.078,179.969,7.603,149.442
C00660=1121.201,73.047,-55.094,179.971,7.607,149.443
C00661=1121.196,73.296,-55.112,179.972,7.611,149.443
C00662=1121.191,73.546,-55.130,179.973,7.614,149.444
C00663=1121.186,73.794,-55.147,179.975,7.618,149.444
C00664=1121.181,74.044,-55.164,179.976,7.622,149.445
C00665=1121.176,74.293,-55.182,179.977,7.626,149.445
C00666=1121.171,74.543,-55.199,179.979,7.630,149.446
C00667=1121.167,74.792,-55.217,179.981,7.634,149.446
C00668=1121.162,75.041,-55.235,179.982,7.638,149.447
C00669=1121.158,75.256,-55.249,179.983,7.642,149.447
C00670=1121.153,75.471,-55.265,179.985,7.645,149.447
C00671=1121.149,75.685,-55.280,179.986,7.648,149.448
C00672=1121.145,75.900,-55.294,179.987,7.652,149.448
C00673=1121.141,76.114,-55.310,179.988,7.655,149.449
C00674=1121.137,76.329,-55.325,179.990,7.659,149.449
C00675=1121.132,76.543,-55.340,179.991,7.662,149.450
C00676=1121.128,76.758,-55.355,179.992,7.665,149.450
C00677=1121.123,77.008,-55.373,179.993,7.669,149.451
C00678=1121.118,77.257,-55.391,179.994,7.673,149.451
C00679=1121.114,77.506,-55.407,179.995,7.677,149.452
C00680=1121.109,77.755,-55.425,179.996,7.680,149.452
C00681=1121.104,78.005,-55.443,179.997,7.684,149.453
C00682=1121.099,78.254,-55.461,179.997,7.688,149.453
C00683=1121.094,78.504,-55.479,179.999,7.692,149.454
C00684=1121.089,78.753,-55.497,180.000,7.695,149.454
C00685=1121.084,79.002,-55.513,-179.999,7.699,149.455
C00686=1121.079,79.251,-55.531,-179.998,7.702,149.456
C00687=1121.074,79.501,-55.549,-179.997,7.706,149.456
C00688=1121.069,79.750,-55.567,-179.996,7.710,149.457
C00689=1121.064,80.000,-55.585,-179.995,7.714,149.457
C00690=1121.059,80.249,-55.602,-179.994,7.717,149.458
C00691=1121.054,80.498,-55.620,-179.993,7.721,149.458
C00692=1121.050,80.747,-55.638,-179.992,7.725,149.459
C00693=1121.045,80.996,-55.656,-179.991,7.729,149.459
C00694=1121.040,81.246,-55.673,-179.990,7.732,149.460
C00695=1121.036,81.496,-55.691,-179.988,7.736,149.460
C00696=1121.031,81.745,-55.709,-179.987,7.740,149.461
C00697=1121.026,81.994,-55.727,-179.986,7.743,149.461
C00698=1121.021,82.243,-55.745,-179.985,7.748,149.462
C00699=1121.016,82.493,-55.763,-179.984,7.751,149.462
C00700=1121.011,82.742,-55.781,-179.983,7.755,149.463
C00701=1121.006,82.991,-55.799,-179.982,7.759,149.463
C00702=1121.001,83.240,-55.817,-179.981,7.762,149.464
C00703=1120.996,83.490,-55.835,-179.979,7.766,149.465
C00704=1120.991,83.739,-55.853,-179.978,7.770,149.465
C00705=1120.986,83.988,-55.871,-179.977,7.774,149.466
C00706=1120.982,84.238,-55.889,-179.976,7.778,149.466
C00707=1120.977,84.487,-55.907,-179.975,7.782,149.467
C00708=1120.972,84.737,-55.924,-179.974,7.785,149.467
C00709=1120.967,84.986,-55.942,-179.972,7.789,149.468
C00710=1120.962,85.235,-55.960,-179.971,7.793,149.468
C00711=1120.957,85.484,-55.978,-179.969,7.797,149.469
C00712=1120.952,85.734,-55.996,-179.968,7.800,149.469
C00713=1120.947,85.983,-56.014,-179.967,7.804,149.470
C00714=1120.943,86.233,-56.032,-179.966,7.808,149.470
C00715=1120.938,86.482,-56.050,-179.965,7.811,149.471
C00716=1120.933,86.731,-56.068,-179.964,7.816,149.471
C00717=1120.928,86.980,-56.086,-179.962,7.820,149.472
C00718=1120.923,87.229,-56.104,-179.960,7.824,149.472
C00719=1120.918,87.479,-56.123,-179.959,7.828,149.473
C00720=1120.913,87.729,-56.141,-179.958,7.831,149.473
C00721=1120.909,87.977,-56.160,-179.957,7.835,149.474
C00722=1120.904,88.226,-56.178,-179.956,7.839,149.474
C00723=1120.899,88.476,-56.196,-179.954,7.843,149.475
C00724=1120.894,88.725,-56.214,-179.952,7.847,149.475
C00725=1120.890,88.939,-56.229,-179.951,7.850,149.476
C00726=1120.886,89.154,-56.245,-179.950,7.853,149.476
C00727=1120.881,89.369,-56.261,-179.949,7.857,149.476
C00728=1120.877,89.583,-56.277,-179.948,7.860,149.477
C00729=1120.873,89.797,-56.293,-179.947,7.863,149.477
C00730=1120.869,90.012,-56.308,-179.945,7.867,149.477
C00731=1120.865,90.227,-56.324,-179.944,7.870,149.478
C00732=1120.861,90.441,-56.340,-179.943,7.873,149.478
C00733=1120.856,90.690,-56.358,-179.941,7.877,149.479
C00734=1120.851,90.940,-56.376,-179.940,7.881,149.479
C00735=1120.846,91.189,-56.394,-179.939,7.885,149.480
C00736=1120.842,91.439,-56.413,-179.937,7.889,149.480
C00737=1120.837,91.687,-56.431,-179.935,7.893,149.481
C00738=1120.831,91.937,-56.450,-179.934,7.897,149.481
C00739=1120.826,92.186,-56.468,-179.932,7.901,149.482
C00740=1120.822,92.436,-56.486,-179.931,7.904,149.482
C00741=1120.817,92.684,-56.505,-179.930,7.908,149.482
C00742=1120.812,92.934,-56.523,-179.928,7.911,149.483
C00743=1120.807,93.183,-56.541,-179.926,7.915,149.483
C00744=1120.803,93.432,-56.560,-179.925,7.919,149.484
C00745=1120.798,93.681,-56.578,-179.923,7.923,149.484
C00746=1120.792,93.931,-56.597,-179.922,7.927,149.485
C00747=1120.788,94.180,-56.616,-179.920,7.931,149.485
C00748=1120.783,94.429,-56.634,-179.918,7.935,149.485
C00749=1120.778,94.679,-56.653,-179.917,7.939,149.486
C00750=1120.774,94.928,-56.672,-179.915,7.943,149.486
C00751=1120.769,95.177,-56.690,-179.914,7.947,149.487
C00752=1120.763,95.427,-56.708,-179.912,7.950,149.487
C00753=1120.759,95.676,-56.727,-179.910,7.954,149.488
C00754=1120.754,95.925,-56.745,-179.909,7.958,149.488
C00755=1120.749,96.174,-56.765,-179.907,7.962,149.488
C00756=1120.745,96.424,-56.783,-179.906,7.966,149.489
C00757=1120.740,96.672,-56.802,-179.904,7.970,149.489
C00758=1120.734,96.922,-56.820,-179.902,7.975,149.490
C00759=1120.730,97.171,-56.839,-179.900,7.978,149.490
C00760=1120.725,97.420,-56.857,-179.898,7.982,149.490
C00761=1120.720,97.669,-56.877,-179.897,7.986,149.491
C00762=1120.716,97.919,-56.895,-179.895,7.990,149.491
C00763=1120.710,98.168,-56.914,-179.893,7.994,149.492
C00764=1120.706,98.418,-56.932,-179.892,7.997,149.492
C00765=1120.701,98.667,-56.952,-179.890,8.001,149.492
C00766=1120.696,98.916,-56.970,-179.888,8.005,149.493
C00767=1120.692,99.165,-56.989,-179.886,8.009,149.493
C00768=1120.686,99.415,-57.007,-179.884,8.013,149.494
C00769=1120.682,99.664,-57.026,-179.882,8.017,149.494
C00770=1120.677,99.913,-57.046,-179.881,8.021,149.494
C00771=1120.672,100.162,-57.064,-179.879,8.025,149.495
C00772=1120.667,100.412,-57.083,-179.877,8.029,149.495
C00773=1120.662,100.661,-57.101,-179.875,8.032,149.495
C00774=1120.658,100.910,-57.121,-179.874,8.036,149.496
C00775=1120.653,101.159,-57.140,-179.871,8.040,149.496
C00776=1120.648,101.409,-57.159,-179.869,8.044,149.496
C00777=1120.643,101.658,-57.177,-179.868,8.048,149.497
C00778=1120.639,101.907,-57.197,-179.866,8.052,149.497
C00779=1120.634,102.156,-57.216,-179.864,8.055,149.497
C00780=1120.628,102.405,-57.234,-179.861,8.060,149.498
C00781=1120.624,102.620,-57.251,-179.861,8.063,149.498
C00782=1120.621,102.834,-57.267,-179.858,8.066,149.498
C00783=1120.617,103.049,-57.284,-179.857,8.069,149.499
C00784=1120.612,103.263,-57.300,-179.855,8.073,149.499
C00785=1120.608,103.477,-57.317,-179.853,8.076,149.499
C00786=1120.604,103.691,-57.333,-179.852,8.079,149.499
C00787=1120.599,103.906,-57.350,-179.850,8.083,149.500
C00788=1120.596,104.121,-57.366,-179.848,8.087,149.500
C00789=1120.591,104.370,-57.385,-179.846,8.090,149.500
C00790=1120.587,104.619,-57.405,-179.845,8.094,149.501
C00791=1120.581,104.868,-57.423,-179.843,8.097,149.501
C00792=1120.576,105.118,-57.443,-179.840,8.102,149.501
C00793=1120.572,105.366,-57.461,-179.838,8.106,149.502
C00794=1120.567,105.616,-57.481,-179.836,8.109,149.502
C00795=1120.562,105.865,-57.500,-179.834,8.113,149.502
C00796=1120.558,106.114,-57.519,-179.832,8.117,149.503
C00797=1120.552,106.363,-57.539,-179.830,8.121,149.503
C00798=1120.547,106.613,-57.558,-179.828,8.124,149.503
C00799=1120.543,106.862,-57.577,-179.826,8.129,149.503
C00800=1120.538,107.111,-57.597,-179.823,8.132,149.504
C00801=1120.533,107.360,-57.616,-179.821,8.136,149.504
C00802=1120.528,107.609,-57.636,-179.819,8.140,149.504
C00803=1120.524,107.858,-57.655,-179.817,8.144,149.504
C00804=1120.519,108.108,-57.674,-179.815,8.148,149.505
C00805=1120.514,108.357,-57.694,-179.812,8.152,149.505
C00806=1120.509,108.606,-57.713,-179.810,8.155,149.505
C00807=1120.505,108.855,-57.732,-179.808,8.159,149.505
C00808=1120.500,109.104,-57.752,-179.806,8.163,149.506
C00809=1120.495,109.354,-57.771,-179.804,8.167,149.506
C00810=1120.490,109.603,-57.791,-179.801,8.170,149.506
C00811=1120.485,109.852,-57.810,-179.799,8.174,149.506
C00812=1120.481,110.102,-57.829,-179.797,8.178,149.507
C00813=1120.476,110.351,-57.849,-179.795,8.183,149.507
C00814=1120.471,110.600,-57.869,-179.792,8.186,149.507
C00815=1120.466,110.849,-57.889,-179.790,8.190,149.507
C00816=1120.461,111.098,-57.908,-179.788,8.193,149.508
C00817=1120.456,111.348,-57.928,-179.786,8.197,149.508
C00818=1120.452,111.597,-57.947,-179.784,8.200,149.508
C00819=1120.447,111.845,-57.967,-179.783,8.204,149.508
C00820=1120.443,112.095,-57.986,-179.781,8.207,149.509
C00821=1120.438,112.344,-58.006,-179.778,8.211,149.509
C00822=1120.433,112.593,-58.025,-179.776,8.214,149.509
C00823=1120.428,112.842,-58.046,-179.775,8.218,149.510
C00824=1120.423,113.092,-58.065,-179.773,8.221,149.510
C00825=1120.418,113.340,-58.085,-179.771,8.225,149.510
C00826=1120.413,113.590,-58.104,-179.769,8.228,149.510
C00827=1120.409,113.839,-58.125,-179.768,8.232,149.511
C00828=1120.404,114.089,-58.144,-179.766,8.235,149.511
C00829=1120.399,114.337,-58.164,-179.763,8.239,149.511
C00830=1120.394,114.586,-58.184,-179.761,8.242,149.511
C00831=1120.390,114.836,-58.204,-179.760,8.246,149.512
C00832=1120.385,115.086,-58.223,-179.758,8.249,149.512
C00833=1120.380,115.334,-58.243,-179.756,8.253,149.512
C00834=1120.375,115.583,-58.263,-179.754,8.256,149.512
C00835=1120.371,115.832,-58.283,-179.753,8.260,149.513
C00836=1120.366,116.082,-58.303,-179.751,8.263,149.513
C00837=1120.361,116.296,-58.320,-179.749,8.266,149.513
C00838=1120.357,116.510,-58.337,-179.748,8.269,149.514
C00839=1120.354,116.724,-58.354,-179.746,8.272,149.514
C00840=1120.350,116.939,-58.371,-179.744,8.275,149.514
C00841=1120.345,117.152,-58.388,-179.743,8.278,149.514
C00842=1120.341,117.368,-58.405,-179.741,8.281,149.514
C00843=1120.337,117.581,-58.423,-179.740,8.283,149.515
C00844=1120.333,117.796,-58.440,-179.738,8.287,149.515
C00845=1120.328,118.045,-58.460,-179.737,8.290,149.515
C00846=1120.323,118.294,-58.480,-179.735,8.293,149.516
C00847=1120.319,118.543,-58.500,-179.733,8.297,149.516
C00848=1120.314,118.793,-58.520,-179.731,8.300,149.516
C00849=1120.310,119.042,-58.540,-179.729,8.304,149.516
C00850=1120.304,119.292,-58.560,-179.728,8.307,149.517
C00851=1120.299,119.540,-58.580,-179.726,8.310,149.517
C00852=1120.295,119.789,-58.601,-179.723,8.314,149.517
C00853=1120.290,120.038,-58.620,-179.721,8.317,149.517
C00854=1120.286,120.287,-58.641,-179.720,8.321,149.518
C00855=1120.281,120.537,-58.660,-179.718,8.324,149.518
C00856=1120.276,120.786,-58.681,-179.716,8.328,149.518
C00857=1120.271,121.035,-58.702,-179.714,8.331,149.518
C00858=1120.266,121.284,-58.721,-179.713,8.334,149.519
C00859=1120.261,121.533,-58.741,-179.711,8.338,149.519
C00860=1120.257,121.782,-58.762,-179.709,8.341,149.519
C00861=1120.252,122.031,-58.781,-179.707,8.345,149.520
C00862=1120.247,122.281,-58.802,-179.706,8.347,149.520
C00863=1120.243,122.530,-58.823,-179.704,8.351,149.520
C00864=1120.238,122.779,-58.842,-179.702,8.355,149.520
C00865=1120.233,123.028,-58.863,-179.700,8.357,149.521
C00866=1120.229,123.277,-58.883,-179.698,8.361,149.521
C00867=1120.224,123.526,-58.904,-179.697,8.365,149.521
C00868=1120.219,123.776,-58.924,-179.695,8.368,149.522
C00869=1120.215,124.025,-58.944,-179.693,8.371,149.522
C00870=1120.210,124.273,-58.964,-179.691,8.374,149.522
C00871=1120.204,124.522,-58.985,-179.689,8.378,149.522
C00872=1120.200,124.771,-59.005,-179.688,8.381,149.523
C00873=1120.195,125.021,-59.025,-179.686,8.385,149.523
C00874=1120.191,125.270,-59.045,-179.684,8.388,149.523
C00875=1120.186,125.519,-59.066,-179.683,8.391,149.523
C00876=1120.181,125.768,-59.087,-179.681,8.395,149.524
C00877=1120.177,126.017,-59.107,-179.679,8.398,149.524
C00878=1120.172,126.266,-59.128,-179.677,8.402,149.524
C00879=1120.167,126.515,-59.148,-179.675,8.404,149.524
C00880=1120.162,126.765,-59.168,-179.674,8.408,149.525
C00881=1120.157,127.014,-59.189,-179.672,8.412,149.525
C00882=1120.153,127.263,-59.209,-179.670,8.414,149.525
C00883=1120.148,127.512,-59.230,-179.668,8.418,149.526
C00884=1120.143,127.761,-59.251,-179.667,8.422,149.526
C00885=1120.139,128.010,-59.271,-179.665,8.425,149.526
C00886=1120.134,128.259,-59.292,-179.663,8.428,149.526
C00887=1120.129,128.508,-59.313,-179.661,8.432,149.527
C00888=1120.125,128.757,-59.333,-179.660,8.435,149.527
C00889=1120.120,129.007,-59.354,-179.658,8.438,149.527
C00890=1120.115,129.256,-59.374,-179.656,8.442,149.528
C00891=1120.110,129.505,-59.395,-179.654,8.444,149.528
C00892=1120.106,129.754,-59.416,-179.653,8.448,149.528
C00893=1120.102,129.968,-59.433,-179.651,8.451,149.528
C00894=1120.097,130.182,-59.451,-179.650,8.454,149.529
C00895=1120.093,130.397,-59.469,-179.648,8.456,149.529
C00896=1120.090,130.611,-59.487,-179.647,8.459,149.529
C00897=1120.085,130.825,-59.504,-179.645,8.463,149.529
C00898=1120.082,131.040,-59.522,-179.643,8.465,149.530
C00899=1120.077,131.253,-59.541,-179.642,8.468,149.530
C00900=1120.073,131.468,-59.559,-179.641,8.471,149.530
C00901=1120.069,131.717,-59.579,-179.639,8.475,149.530
C00902=1120.064,131.966,-59.600,-179.637,8.477,149.531
C00903=1120.059,132.215,-59.620,-179.635,8.481,149.531
C00904=1120.054,132.464,-59.641,-179.634,8.484,149.531
C00905=1120.050,132.713,-59.662,-179.632,8.487,149.532
C00906=1120.045,132.962,-59.683,-179.630,8.491,149.532
C00907=1120.040,133.211,-59.704,-179.629,8.494,149.532
C00908=1120.035,133.460,-59.725,-179.627,8.497,149.532
C00909=1120.031,133.710,-59.746,-179.625,8.501,149.533
C00910=1120.026,133.959,-59.766,-179.624,8.504,149.533
C00911=1120.021,134.208,-59.787,-179.622,8.508,149.533
C00912=1120.017,134.456,-59.808,-179.621,8.510,149.534
C00913=1120.012,134.706,-59.829,-179.619,8.514,149.534
C00914=1120.007,134.955,-59.850,-179.617,8.518,149.534
C00915=1120.002,135.204,-59.871,-179.615,8.520,149.534
C00916=1119.998,135.453,-59.893,-179.614,8.524,149.535
C00917=1119.993,135.702,-59.913,-179.612,8.527,149.535
C00918=1119.988,135.951,-59.934,-179.610,8.530,149.535
C00919=1119.983,136.200,-59.956,-179.609,8.534,149.536
C00920=1119.979,136.449,-59.976,-179.607,8.537,149.536
C00921=1119.974,136.698,-59.997,-179.605,8.540,149.536
C00922=1119.970,136.947,-60.019,-179.604,8.544,149.537
C00923=1119.965,137.196,-60.040,-179.602,8.547,149.537
C00924=1119.960,137.446,-60.061,-179.600,8.551,149.537
C00925=1119.956,137.694,-60.082,-179.599,8.554,149.538
C00926=1119.951,137.943,-60.103,-179.597,8.557,149.538
C00927=1119.946,138.193,-60.124,-179.596,8.560,149.538
C00928=1119.942,138.442,-60.145,-179.594,8.564,149.538
C00929=1119.937,138.691,-60.166,-179.592,8.568,149.539
C00930=1119.932,138.939,-60.188,-179.591,8.570,149.539
C00931=1119.927,139.188,-60.208,-179.589,8.574,149.539
C00932=1119.923,139.438,-60.230,-179.588,8.577,149.540
C00933=1119.918,139.687,-60.251,-179.586,8.580,149.540
C00934=1119.913,139.936,-60.272,-179.584,8.584,149.540
C00935=1119.909,140.185,-60.293,-179.582,8.587,149.541
C00936=1119.904,140.435,-60.314,-179.581,8.591,149.541
C00937=1119.899,140.683,-60.336,-179.579,8.594,149.541
C00938=1119.894,140.933,-60.357,-179.578,8.597,149.542
C00939=1119.890,141.181,-60.378,-179.576,8.600,149.542
C00940=1119.885,141.431,-60.399,-179.575,8.604,149.542
C00941=1119.880,141.679,-60.421,-179.573,8.607,149.543
C00942=1119.875,141.929,-60.442,-179.572,8.611,149.543
C00943=1119.871,142.177,-60.463,-179.570,8.614,149.543
C00944=1119.867,142.426,-60.485,-179.569,8.617,149.544
C00945=1119.862,142.676,-60.506,-179.566,8.621,149.544
C00946=1119.857,142.924,-60.528,-179.565,8.624,149.544
C00947=1119.852,143.174,-60.549,-179.563,8.627,149.545
C00948=1119.848,143.423,-60.570,-179.562,8.631,149.545
C00949=1119.844,143.637,-60.589,-179.560,8.634,149.545
C00950=1119.840,143.851,-60.607,-179.559,8.637,149.546
C00951=1119.836,144.065,-60.626,-179.558,8.640,149.546
C00952=1119.831,144.280,-60.644,-179.556,8.642,149.546
C00953=1119.828,144.493,-60.663,-179.555,8.645,149.547
C00954=1119.823,144.707,-60.682,-179.554,8.648,149.547
C00955=1119.820,144.921,-60.699,-179.552,8.651,149.547
C00956=1119.816,145.136,-60.718,-179.551,8.654,149.548
C00957=1119.811,145.384,-60.740,-179.549,8.658,149.548
C00958=1119.805,145.633,-60.761,-179.547,8.662,149.548
C00959=1119.802,145.882,-60.782,-179.544,8.666,149.548
C00960=1119.797,146.131,-60.804,-179.542,8.669,149.548
C00961=1119.793,146.380,-60.826,-179.540,8.673,149.549
C00962=1119.788,146.630,-60.847,-179.537,8.677,149.549
C00963=1119.783,146.878,-60.869,-179.535,8.681,149.549
C00964=1119.779,147.128,-60.891,-179.532,8.685,149.549
C00965=1119.774,147.376,-60.913,-179.530,8.688,149.549
C00966=1119.769,147.625,-60.934,-179.528,8.692,149.550
C00967=1119.764,147.875,-60.956,-179.525,8.696,149.550
C00968=1119.759,148.124,-60.977,-179.523,8.699,149.550
C00969=1119.755,148.373,-60.999,-179.521,8.703,149.550
C00970=1119.750,148.622,-61.021,-179.518,8.707,149.551
C00971=1119.745,148.870,-61.043,-179.516,8.711,149.551
C00972=1119.741,149.120,-61.065,-179.513,8.714,149.551
C00973=1119.736,149.368,-61.086,-179.511,8.718,149.551
C00974=1119.732,149.618,-61.108,-179.509,8.721,149.551
C00975=1119.727,149.867,-61.129,-179.507,8.725,149.552
C00976=1119.722,150.116,-61.151,-179.504,8.729,149.552
C00977=1119.718,150.365,-61.173,-179.501,8.732,149.552
C00978=1119.713,150.613,-61.195,-179.499,8.736,149.552
C00979=1119.708,150.863,-61.217,-179.497,8.739,149.552
C00980=1119.703,151.112,-61.239,-179.495,8.743,149.553
C00981=1119.699,151.361,-61.261,-179.492,8.747,149.553
C00982=1119.694,151.610,-61.283,-179.490,8.750,149.553
C00983=1119.689,151.859,-61.305,-179.488,8.754,149.553
C00984=1119.685,152.108,-61.327,-179.485,8.758,149.553
C00985=1119.680,152.357,-61.349,-179.483,8.761,149.553
C00986=1119.676,152.605,-61.371,-179.481,8.764,149.554
C00987=1119.671,152.854,-61.393,-179.478,8.768,149.554
C00988=1119.666,153.103,-61.415,-179.476,8.771,149.554
C00989=1119.662,153.353,-61.437,-179.473,8.775,149.554
C00990=1119.657,153.601,-61.459,-179.471,8.779,149.554
C00991=1119.652,153.851,-61.481,-179.469,8.782,149.554
C00992=1119.648,154.099,-61.503,-179.467,8.785,149.555
C00993=1119.643,154.349,-61.526,-179.464,8.788,149.555
C00994=1119.638,154.597,-61.548,-179.462,8.792,149.555
C00995=1119.634,154.846,-61.570,-179.460,8.795,149.555
C00996=1119.629,155.096,-61.592,-179.457,8.799,149.555
C00997=1119.624,155.345,-61.614,-179.455,8.803,149.555
C00998=1119.620,155.593,-61.637,-179.452,8.806,149.555
C00999=1119.615,155.842,-61.659,-179.450,8.809,149.556
C01000=1119.611,156.091,-61.681,-179.448,8.813,149.556
C01001=1119.605,156.340,-61.703,-179.445,8.816,149.556
C01002=1119.601,156.589,-61.726,-179.443,8.820,149.556
C01003=1119.597,156.838,-61.748,-179.441,8.823,149.556
C01004=1119.592,157.087,-61.770,-179.439,8.826,149.556
C01005=1119.588,157.301,-61.789,-179.436,8.829,149.556
C01006=1119.584,157.515,-61.808,-179.435,8.832,149.557
C01007=1119.580,157.729,-61.828,-179.432,8.835,149.557
C01008=1119.576,157.943,-61.847,-179.430,8.837,149.557
C01009=1119.572,158.157,-61.866,-179.428,8.841,149.557
C01010=1119.568,158.371,-61.886,-179.426,8.843,149.557
C01011=1119.564,158.585,-61.905,-179.424,8.847,149.557
C01012=1119.560,158.799,-61.924,-179.422,8.849,149.557
C01013=1119.556,159.048,-61.946,-179.420,8.852,149.557
C01014=1119.550,159.297,-61.969,-179.418,8.856,149.557
C01015=1119.546,159.546,-61.991,-179.415,8.859,149.558
C01016=1119.542,159.795,-62.014,-179.413,8.862,149.558
C01017=1119.537,160.043,-62.037,-179.411,8.865,149.558
C01018=1119.533,160.293,-62.059,-179.409,8.869,149.558
C01019=1119.528,160.542,-62.082,-179.406,8.872,149.558
C01020=1119.523,160.790,-62.104,-179.404,8.875,149.558
C01021=1119.519,161.039,-62.126,-179.401,8.878,149.558
C01022=1119.514,161.289,-62.149,-179.399,8.882,149.558
C01023=1119.510,161.537,-62.171,-179.397,8.885,149.559
C01024=1119.505,161.786,-62.194,-179.394,8.888,149.559
C01025=1119.501,162.035,-62.217,-179.392,8.892,149.559
C01026=1119.496,162.285,-62.239,-179.390,8.895,149.559
C01027=1119.491,162.533,-62.262,-179.387,8.898,149.559
C01028=1119.486,162.782,-62.285,-179.385,8.901,149.559
C01029=1119.482,163.031,-62.307,-179.383,8.904,149.559
C01030=1119.477,163.279,-62.330,-179.380,8.908,149.559
C01031=1119.472,163.529,-62.352,-179.379,8.910,149.559
C01032=1119.468,163.778,-62.376,-179.376,8.913,149.560
C01033=1119.464,164.026,-62.398,-179.374,8.917,149.560
C01034=1119.459,164.276,-62.421,-179.371,8.920,149.560
C01035=1119.454,164.524,-62.443,-179.369,8.923,149.560
C01036=1119.450,164.773,-62.467,-179.367,8.927,149.560
C01037=1119.446,165.022,-62.490,-179.364,8.930,149.560
C01038=1119.441,165.272,-62.512,-179.362,8.933,149.560
C01039=1119.435,165.520,-62.535,-179.360,8.936,149.560
C01040=1119.431,165.769,-62.558,-179.358,8.939,149.560
C01041=1119.427,166.018,-62.581,-179.355,8.942,149.560
C01042=1119.422,166.267,-62.603,-179.353,8.945,149.561
C01043=1119.418,166.516,-62.627,-179.351,8.948,149.561
C01044=1119.412,166.764,-62.650,-179.348,8.951,149.561
C01045=1119.408,167.013,-62.673,-179.346,8.955,149.561
C01046=1119.404,167.262,-62.696,-179.344,8.957,149.561
C01047=1119.399,167.512,-62.719,-179.342,8.960,149.561
C01048=1119.395,167.760,-62.741,-179.340,8.964,149.561
C01049=1119.389,168.009,-62.764,-179.337,8.967,149.561
C01050=1119.385,168.258,-62.788,-179.335,8.970,149.561
C01051=1119.381,168.507,-62.810,-179.333,8.973,149.562
C01052=1119.376,168.756,-62.834,-179.331,8.976,149.562
C01053=1119.371,169.005,-62.857,-179.328,8.979,149.562
C01054=1119.367,169.253,-62.880,-179.325,8.982,149.562
C01055=1119.362,169.503,-62.903,-179.324,8.985,149.562
C01056=1119.357,169.751,-62.926,-179.321,8.988,149.562
C01057=1119.352,170.000,-62.949,-179.319,8.991,149.562
C01058=1119.348,170.249,-62.972,-179.317,8.995,149.562
C01059=1119.344,170.498,-62.995,-179.314,8.998,149.562
C01060=1119.339,170.747,-63.018,-179.312,9.000,149.562
C01061=1119.335,170.961,-63.038,-179.310,9.003,149.563
C01062=1119.331,171.174,-63.058,-179.308,9.006,149.563
C01063=1119.327,171.388,-63.078,-179.307,9.008,149.563
C01064=1119.324,171.602,-63.099,-179.305,9.010,149.563
C01065=1119.320,171.816,-63.118,-179.303,9.013,149.563
C01066=1119.315,172.030,-63.138,-179.301,9.016,149.563
C01067=1119.311,172.244,-63.158,-179.299,9.019,149.563
C01068=1119.308,172.458,-63.178,-179.297,9.021,149.563
C01069=1119.303,172.707,-63.201,-179.295,9.024,149.563
C01070=1119.298,172.956,-63.224,-179.293,9.027,149.563
C01071=1119.294,173.204,-63.248,-179.290,9.030,149.563
C01072=1119.289,173.453,-63.272,-179.288,9.033,149.564
C01073=1119.285,173.702,-63.295,-179.286,9.036,149.564
C01074=1119.280,173.951,-63.318,-179.284,9.039,149.564
C01075=1119.276,174.200,-63.341,-179.281,9.042,149.564
C01076=1119.271,174.449,-63.365,-179.279,9.045,149.564
C01077=1119.267,174.697,-63.389,-179.277,9.048,149.564
C01078=1119.262,174.946,-63.412,-179.275,9.051,149.564
C01079=1119.257,175.195,-63.435,-179.273,9.054,149.564
C01080=1119.253,175.444,-63.459,-179.271,9.057,149.564
C01081=1119.248,175.689,-63.481,-179.268,9.060,149.564
C01082=1119.244,175.935,-63.505,-179.267,9.062,149.565
C01083=1119.240,176.180,-63.528,-179.264,9.066,149.565
C01084=1119.234,176.425,-63.551,-179.262,9.069,149.565
C01085=1119.231,176.670,-63.575,-179.260,9.071,149.565
C01086=1119.226,176.916,-63.598,-179.258,9.074,149.565
C01087=1119.221,177.161,-63.620,-179.256,9.077,149.565
C01088=1119.217,177.406,-63.644,-179.253,9.080,149.565
C01089=1119.212,177.655,-63.668,-179.251,9.083,149.565
C01090=1119.208,177.904,-63.691,-179.249,9.086,149.565
C01091=1119.203,178.153,-63.715,-179.247,9.089,149.565
C01092=1119.199,178.402,-63.739,-179.245,9.092,149.566
C01093=1119.194,178.651,-63.762,-179.243,9.095,149.566
C01094=1119.190,178.899,-63.786,-179.241,9.098,149.566
C01095=1119.185,179.148,-63.809,-179.239,9.100,149.566
C01096=1119.180,179.396,-63.833,-179.236,9.104,149.566
C01097=1119.176,179.646,-63.857,-179.233,9.107,149.566
C01098=1119.171,179.895,-63.880,-179.231,9.111,149.566
C01099=1119.167,180.143,-63.904,-179.228,9.114,149.566
C01100=1119.163,180.393,-63.928,-179.226,9.117,149.566
C01101=1119.158,180.641,-63.952,-179.223,9.120,149.566
C01102=1119.153,180.890,-63.975,-179.220,9.124,149.566
C01103=1119.149,181.139,-63.999,-179.217,9.126,149.566
C01104=1119.144,181.388,-64.023,-179.215,9.130,149.566
C01105=1119.140,181.636,-64.047,-179.212,9.133,149.566
C01106=1119.135,181.885,-64.070,-179.210,9.136,149.566
C01107=1119.131,182.133,-64.094,-179.207,9.139,149.566
C01108=1119.125,182.383,-64.118,-179.205,9.142,149.566
C01109=1119.122,182.632,-64.143,-179.202,9.145,149.566
C01110=1119.117,182.880,-64.167,-179.199,9.148,149.566
C01111=1119.113,183.129,-64.190,-179.197,9.151,149.566
C01112=1119.108,183.378,-64.214,-179.194,9.154,149.566
C01113=1119.104,183.626,-64.238,-179.191,9.157,149.566
C01114=1119.098,183.876,-64.262,-179.189,9.160,149.566
C01115=1119.095,184.125,-64.287,-179.186,9.163,149.566
C01116=1119.090,184.374,-64.310,-179.184,9.167,149.566
C01117=1119.086,184.591,-64.331,-179.182,9.169,149.566
C01118=1119.082,184.808,-64.352,-179.180,9.171,149.566
C01119=1119.078,185.025,-64.373,-179.178,9.174,149.566
C01120=1119.074,185.243,-64.394,-179.175,9.176,149.566
C01121=1119.070,185.460,-64.415,-179.173,9.179,149.566
C01122=1119.066,185.677,-64.436,-179.171,9.182,149.566
C01123=1119.063,185.894,-64.458,-179.169,9.184,149.566
C01124=1119.058,186.112,-64.479,-179.167,9.186,149.566
C01125=1119.053,186.361,-64.503,-179.165,9.189,149.566
C01126=1119.050,186.610,-64.527,-179.162,9.193,149.567
C01127=1119.045,186.859,-64.551,-179.160,9.195,149.567
C01128=1119.040,187.107,-64.575,-179.158,9.198,149.567
C01129=1119.035,187.356,-64.599,-179.155,9.201,149.567
C01130=1119.032,187.605,-64.624,-179.153,9.204,149.567
C01131=1119.026,187.854,-64.649,-179.151,9.207,149.567
C01132=1119.022,188.103,-64.672,-179.148,9.210,149.567
C01133=1119.017,188.351,-64.696,-179.146,9.212,149.567
C01134=1119.013,188.601,-64.721,-179.144,9.215,149.567
C01135=1119.008,188.849,-64.745,-179.141,9.218,149.567
C01136=1119.004,189.097,-64.769,-179.139,9.221,149.567
C01137=1118.999,189.346,-64.794,-179.137,9.224,149.567
C01138=1118.995,189.595,-64.818,-179.135,9.226,149.567
C01139=1118.991,189.844,-64.842,-179.132,9.229,149.567
C01140=1118.986,190.092,-64.867,-179.130,9.231,149.567
C01141=1118.981,190.341,-64.891,-179.128,9.235,149.567
C01142=1118.977,190.590,-64.916,-179.126,9.237,149.567
C01143=1118.972,190.839,-64.940,-179.124,9.240,149.567
C01144=1118.968,191.087,-64.964,-179.122,9.242,149.567
C01145=1118.963,191.336,-64.989,-179.119,9.245,149.567
C01146=1118.959,191.585,-65.013,-179.117,9.248,149.567
C01147=1118.954,191.834,-65.038,-179.115,9.251,149.568
C01148=1118.950,192.083,-65.062,-179.113,9.254,149.568
C01149=1118.945,192.331,-65.087,-179.111,9.256,149.568
C01150=1118.940,192.580,-65.111,-179.109,9.259,149.568
C01151=1118.936,192.829,-65.136,-179.107,9.261,149.568
C01152=1118.932,193.078,-65.160,-179.105,9.265,149.568
C01153=1118.926,193.326,-65.185,-179.103,9.267,149.568
C01154=1118.923,193.575,-65.209,-179.101,9.269,149.568
C01155=1118.917,193.824,-65.234,-179.098,9.273,149.568
C01156=1118.913,194.073,-65.258,-179.097,9.275,149.568
C01157=1118.909,194.321,-65.284,-179.095,9.278,149.568
C01158=1118.904,194.570,-65.308,-179.093,9.281,149.569
C01159=1118.900,194.819,-65.333,-179.091,9.283,149.569
C01160=1118.896,195.068,-65.357,-179.089,9.286,149.569
C01161=1118.890,195.316,-65.382,-179.088,9.288,149.569
C01162=1118.887,195.565,-65.406,-179.085,9.292,149.569
C01163=1118.882,195.814,-65.432,-179.084,9.294,149.569
C01164=1118.877,196.062,-65.456,-179.082,9.297,149.569
C01165=1118.873,196.311,-65.481,-179.080,9.299,149.570
C01166=1118.868,196.560,-65.505,-179.077,9.303,149.569
C01167=1118.864,196.809,-65.530,-179.074,9.306,149.569
C01168=1118.859,197.057,-65.555,-179.071,9.309,149.569
C01169=1118.855,197.306,-65.580,-179.068,9.313,149.569
C01170=1118.850,197.555,-65.604,-179.065,9.316,149.569
C01171=1118.846,197.803,-65.629,-179.061,9.320,149.569
C01172=1118.842,198.052,-65.654,-179.058,9.323,149.569
C01173=1118.838,198.266,-65.676,-179.056,9.326,149.569
C01174=1118.834,198.480,-65.697,-179.053,9.329,149.569
C01175=1118.830,198.694,-65.718,-179.051,9.332,149.569
C01176=1118.826,198.907,-65.739,-179.048,9.334,149.569
C01177=1118.822,199.121,-65.761,-179.045,9.337,149.569
C01178=1118.819,199.335,-65.782,-179.042,9.340,149.569
C01179=1118.815,199.548,-65.803,-179.039,9.343,149.569
C01180=1118.811,199.762,-65.825,-179.037,9.345,149.569
C01181=1118.806,200.010,-65.850,-179.034,9.349,149.569
C01182=1118.802,200.259,-65.875,-179.031,9.352,149.568
C01183=1118.797,200.507,-65.900,-179.028,9.355,149.569
C01184=1118.793,200.757,-65.925,-179.025,9.358,149.568
C01185=1118.788,201.005,-65.951,-179.022,9.361,149.568
C01186=1118.784,201.254,-65.976,-179.018,9.364,149.568
C01187=1118.779,201.502,-66.000,-179.015,9.367,149.568
C01188=1118.775,201.751,-66.025,-179.013,9.370,149.568
C01189=1118.771,202.000,-66.051,-179.010,9.373,149.568
C01190=1118.766,202.248,-66.077,-179.006,9.377,149.568
C01191=1118.762,202.497,-66.101,-179.003,9.379,149.568
C01192=1118.757,202.746,-66.126,-179.001,9.382,149.568
C01193=1118.753,202.995,-66.151,-178.998,9.385,149.567
C01194=1118.748,203.243,-66.177,-178.995,9.388,149.567
C01195=1118.744,203.492,-66.202,-178.991,9.391,149.567
C01196=1118.739,203.741,-66.228,-178.988,9.394,149.567
C01197=1118.735,203.989,-66.252,-178.986,9.397,149.567
C01198=1118.731,204.238,-66.278,-178.983,9.400,149.567
C01199=1118.726,204.487,-66.303,-178.980,9.403,149.567
C01200=1118.721,204.735,-66.328,-178.977,9.405,149.567
C01201=1118.717,204.984,-66.354,-178.974,9.409,149.567
C01202=1118.712,205.233,-66.379,-178.971,9.411,149.567
C01203=1118.708,205.482,-66.405,-178.968,9.414,149.566
C01204=1118.703,205.730,-66.430,-178.965,9.417,149.566
C01205=1118.699,205.979,-66.456,-178.963,9.420,149.566
C01206=1118.695,206.228,-66.482,-178.960,9.423,149.566
C01207=1118.690,206.476,-66.506,-178.957,9.425,149.566
C01208=1118.685,206.725,-66.532,-178.954,9.429,149.566
C01209=1118.681,206.974,-66.558,-178.951,9.431,149.566
C01210=1118.676,207.222,-66.583,-178.949,9.434,149.566
C01211=1118.672,207.471,-66.609,-178.946,9.437,149.566
C01212=1118.668,207.720,-66.635,-178.943,9.440,149.566
C01213=1118.663,207.968,-66.660,-178.941,9.443,149.566
C01214=1118.658,208.217,-66.685,-178.938,9.446,149.566
C01215=1118.654,208.466,-66.711,-178.935,9.448,149.566
C01216=1118.649,208.714,-66.736,-178.932,9.452,149.566
C01217=1118.645,208.963,-66.762,-178.929,9.454,149.565
C01218=1118.641,209.212,-66.788,-178.927,9.457,149.566
C01219=1118.636,209.460,-66.813,-178.925,9.460,149.566
C01220=1118.632,209.708,-66.839,-178.922,9.462,149.565
C01221=1118.628,209.957,-66.865,-178.919,9.466,149.565
C01222=1118.623,210.206,-66.890,-178.916,9.468,149.565
C01223=1118.619,210.454,-66.916,-178.914,9.471,149.565
C01224=1118.614,210.703,-66.941,-178.911,9.475,149.565
C01225=1118.610,210.952,-66.967,-178.909,9.477,149.565
C01226=1118.606,211.201,-66.993,-178.906,9.480,149.565
C01227=1118.601,211.449,-67.018,-178.904,9.483,149.565
C01228=1118.596,211.698,-67.045,-178.901,9.486,149.565
C01229=1118.593,211.911,-67.067,-178.899,9.488,149.566
C01230=1118.590,212.125,-67.089,-178.898,9.491,149.566
C01231=1118.585,212.338,-67.112,-178.895,9.493,149.565
C01232=1118.582,212.552,-67.133,-178.893,9.496,149.565
C01233=1118.577,212.765,-67.156,-178.891,9.498,149.566
C01234=1118.574,212.978,-67.178,-178.889,9.500,149.566
C01235=1118.570,213.192,-67.201,-178.886,9.503,149.566
C01236=1118.566,213.406,-67.222,-178.885,9.506,149.566
C01237=1118.562,213.655,-67.248,-178.883,9.508,149.566
C01238=1118.557,213.903,-67.275,-178.881,9.512,149.566
C01239=1118.553,214.151,-67.300,-178.879,9.514,149.566
C01240=1118.548,214.400,-67.326,-178.877,9.517,149.566
C01241=1118.544,214.649,-67.352,-178.875,9.520,149.566
C01242=1118.540,214.897,-67.378,-178.873,9.523,149.567
C01243=1118.535,215.146,-67.405,-178.871,9.525,149.567
C01244=1118.530,215.394,-67.430,-178.868,9.529,149.567
C01245=1118.526,215.643,-67.456,-178.867,9.531,149.567
C01246=1118.522,215.891,-67.482,-178.864,9.534,149.567
C01247=1118.517,216.141,-67.509,-178.862,9.537,149.567
C01248=1118.513,216.389,-67.534,-178.860,9.540,149.567
C01249=1118.509,216.638,-67.561,-178.858,9.543,149.567
C01250=1118.505,216.886,-67.587,-178.855,9.546,149.567
C01251=1118.500,217.135,-67.613,-178.853,9.549,149.568
C01252=1118.495,217.383,-67.639,-178.851,9.552,149.568
C01253=1118.491,217.632,-67.665,-178.849,9.555,149.568
C01254=1118.486,217.881,-67.691,-178.846,9.558,149.568
C01255=1118.482,218.129,-67.718,-178.844,9.561,149.568
C01256=1118.478,218.378,-67.743,-178.842,9.564,149.568
C01257=1118.473,218.626,-67.770,-178.840,9.567,149.568
C01258=1118.469,218.875,-67.796,-178.837,9.570,149.568
C01259=1118.465,219.124,-67.822,-178.834,9.574,149.568
C01260=1118.460,219.372,-67.849,-178.833,9.576,149.568
C01261=1118.456,219.621,-67.875,-178.830,9.579,149.569
C01262=1118.452,219.869,-67.901,-178.828,9.582,149.569
C01263=1118.447,220.118,-67.927,-178.825,9.586,149.569
C01264=1118.443,220.366,-67.954,-178.823,9.589,149.569
C01265=1118.438,220.615,-67.980,-178.820,9.592,149.569
C01266=1118.434,220.863,-68.007,-178.818,9.595,149.569
C01267=1118.430,221.112,-68.032,-178.815,9.598,149.569
C01268=1118.425,221.361,-68.059,-178.813,9.601,149.569
C01269=1118.421,221.609,-68.085,-178.810,9.604,149.569
C01270=1118.416,221.858,-68.112,-178.808,9.607,149.569
C01271=1118.412,222.106,-68.139,-178.805,9.610,149.569
C01272=1118.407,222.355,-68.165,-178.803,9.614,149.569
C01273=1118.403,222.603,-68.191,-178.800,9.617,149.569
C01274=1118.398,222.853,-68.218,-178.798,9.620,149.570
C01275=1118.394,223.101,-68.244,-178.795,9.623,149.570
C01276=1118.390,223.349,-68.271,-178.793,9.626,149.570
C01277=1118.386,223.598,-68.297,-178.789,9.630,149.570
C01278=1118.381,223.846,-68.324,-178.787,9.633,149.570
C01279=1118.377,224.095,-68.351,-178.784,9.636,149.570
C01280=1118.372,224.343,-68.378,-178.782,9.639,149.570
C01281=1118.368,224.592,-68.403,-178.779,9.642,149.570
C01282=1118.363,224.840,-68.430,-178.776,9.645,149.570
C01283=1118.360,225.089,-68.457,-178.773,9.649,149.570
C01284=1118.355,225.337,-68.484,-178.771,9.652,149.570
C01285=1118.351,225.551,-68.507,-178.768,9.654,149.570
C01286=1118.347,225.764,-68.530,-178.766,9.657,149.570
C01287=1118.344,225.977,-68.552,-178.763,9.660,149.570
C01288=1118.340,226.191,-68.575,-178.761,9.663,149.570
C01289=1118.336,226.404,-68.598,-178.758,9.665,149.570
C01290=1118.332,226.617,-68.622,-178.756,9.668,149.570
C01291=1118.328,226.831,-68.644,-178.754,9.671,149.570
C01292=1118.325,227.045,-68.667,-178.751,9.674,149.570
C01293=1118.321,227.294,-68.694,-178.749,9.677,149.570
C01294=1118.316,227.542,-68.721,-178.745,9.680,149.570
C01295=1118.312,227.790,-68.747,-178.742,9.683,149.570
C01296=1118.307,228.039,-68.775,-178.739,9.686,149.570
C01297=1118.303,228.287,-68.802,-178.736,9.690,149.570
C01298=1118.299,228.535,-68.828,-178.733,9.693,149.570
C01299=1118.294,228.784,-68.855,-178.730,9.696,149.570
C01300=1118.289,229.032,-68.882,-178.727,9.699,149.570
C01301=1118.285,229.282,-68.910,-178.724,9.702,149.570
C01302=1118.281,229.530,-68.936,-178.721,9.706,149.570
C01303=1118.277,229.778,-68.963,-178.718,9.708,149.569
C01304=1118.272,230.027,-68.990,-178.714,9.712,149.569
C01305=1118.268,230.275,-69.017,-178.711,9.715,149.569
C01306=1118.264,230.524,-69.044,-178.708,9.718,149.569
C01307=1118.259,230.772,-69.071,-178.705,9.721,149.569
C01308=1118.255,231.021,-69.098,-178.702,9.724,149.569
C01309=1118.250,231.270,-69.125,-178.699,9.727,149.569
C01310=1118.246,231.518,-69.153,-178.696,9.730,149.569
C01311=1118.242,231.766,-69.180,-178.693,9.733,149.569
C01312=1118.237,232.014,-69.207,-178.690,9.736,149.568
C01313=1118.233,232.263,-69.234,-178.687,9.738,149.568
C01314=1118.229,232.512,-69.261,-178.684,9.741,149.568
C01315=1118.224,232.760,-69.288,-178.680,9.745,149.568
C01316=1118.220,233.008,-69.316,-178.678,9.748,149.568
C01317=1118.216,233.258,-69.343,-178.675,9.751,149.568
C01318=1118.212,233.506,-69.370,-178.672,9.753,149.568
C01319=1118.207,233.754,-69.397,-178.669,9.756,149.568
C01320=1118.203,234.002,-69.425,-178.666,9.759,149.568
C01321=1118.199,234.251,-69.452,-178.663,9.762,149.568
C01322=1118.194,234.500,-69.479,-178.660,9.764,149.567
C01323=1118.190,234.748,-69.507,-178.657,9.767,149.567
C01324=1118.185,234.996,-69.534,-178.654,9.770,149.567
C01325=1118.181,235.245,-69.561,-178.652,9.773,149.567
C01326=1118.176,235.493,-69.589,-178.649,9.775,149.567
C01327=1118.172,235.742,-69.616,-178.646,9.778,149.567
C01328=1118.167,235.990,-69.643,-178.644,9.780,149.567
C01329=1118.163,236.239,-69.671,-178.641,9.783,149.567
C01330=1118.159,236.487,-69.699,-178.638,9.786,149.567
C01331=1118.154,236.735,-69.726,-178.635,9.788,149.567
C01332=1118.150,236.984,-69.754,-178.633,9.791,149.567
C01333=1118.146,237.233,-69.781,-178.630,9.794,149.566
C01334=1118.141,237.481,-69.809,-178.627,9.796,149.566
C01335=1118.137,237.730,-69.836,-178.625,9.798,149.566
C01336=1118.133,237.978,-69.864,-178.622,9.801,149.566
C01337=1118.128,238.226,-69.891,-178.619,9.804,149.566
C01338=1118.125,238.475,-69.919,-178.617,9.806,149.566
C01339=1118.120,238.723,-69.946,-178.614,9.809,149.566
C01340=1118.116,238.971,-69.974,-178.611,9.812,149.566
C01341=1118.112,239.185,-69.998,-178.609,9.814,149.566
C01342=1118.109,239.398,-70.021,-178.607,9.816,149.566
C01343=1118.104,239.611,-70.045,-178.605,9.818,149.566
C01344=1118.100,239.824,-70.069,-178.602,9.820,149.566
C01345=1118.097,240.038,-70.093,-178.601,9.823,149.566
C01346=1118.094,240.251,-70.116,-178.598,9.825,149.566
C01347=1118.089,240.464,-70.140,-178.596,9.827,149.566
C01348=1118.086,240.678,-70.164,-178.594,9.829,149.565
C01349=1118.082,240.926,-70.192,-178.592,9.831,149.565
C01350=1118.077,241.175,-70.219,-178.589,9.834,149.565
C01351=1118.073,241.423,-70.247,-178.587,9.836,149.565
C01352=1118.069,241.671,-70.275,-178.585,9.838,149.565
C01353=1118.064,241.921,-70.303,-178.582,9.841,149.565
C01354=1118.060,242.168,-70.331,-178.580,9.843,149.565
C01355=1118.056,242.417,-70.359,-178.578,9.847,149.565
C01356=1118.052,242.665,-70.387,-178.575,9.849,149.565
C01357=1118.047,242.913,-70.414,-178.573,9.851,149.565
C01358=1118.043,243.162,-70.442,-178.571,9.854,149.565
C01359=1118.038,243.410,-70.470,-178.569,9.856,149.565
C01360=1118.034,243.659,-70.498,-178.567,9.858,149.565
C01361=1118.030,243.907,-70.525,-178.564,9.861,149.565
C01362=1118.026,244.156,-70.554,-178.562,9.863,149.565
C01363=1118.021,244.404,-70.582,-178.560,9.866,149.565
C01364=1118.017,244.652,-70.610,-178.558,9.868,149.565
C01365=1118.012,244.901,-70.637,-178.556,9.870,149.565
C01366=1118.008,245.149,-70.665,-178.554,9.874,149.565
C01367=1118.004,245.398,-70.694,-178.552,9.876,149.565
C01368=1117.999,245.646,-70.721,-178.550,9.878,149.566
C01369=1117.996,245.894,-70.750,-178.548,9.881,149.566
C01370=1117.991,246.142,-70.777,-178.546,9.883,149.566
C01371=1117.987,246.391,-70.806,-178.544,9.886,149.566
C01372=1117.982,246.639,-70.833,-178.542,9.888,149.566
C01373=1117.978,246.888,-70.861,-178.540,9.891,149.566
C01374=1117.973,247.136,-70.890,-178.538,9.893,149.566
C01375=1117.969,247.385,-70.918,-178.536,9.896,149.566
C01376=1117.965,247.633,-70.946,-178.533,9.899,149.566
C01377=1117.961,247.882,-70.974,-178.528,9.903,149.566
C01378=1117.956,248.129,-71.002,-178.523,9.908,149.566
C01379=1117.953,248.378,-71.030,-178.518,9.912,149.565
C01380=1117.947,248.626,-71.059,-178.514,9.916,149.565
C01381=1117.944,248.875,-71.087,-178.510,9.919,149.565
C01382=1117.940,249.123,-71.115,-178.505,9.923,149.564
C01383=1117.935,249.372,-71.143,-178.501,9.926,149.564
C01384=1117.931,249.620,-71.171,-178.496,9.930,149.564
C01385=1117.926,249.868,-71.200,-178.492,9.933,149.564
C01386=1117.922,250.117,-71.228,-178.488,9.936,149.563
C01387=1117.917,250.364,-71.257,-178.484,9.940,149.563
C01388=1117.914,250.613,-71.285,-178.481,9.942,149.563
C01389=1117.909,250.862,-71.314,-178.478,9.945,149.563
C01390=1117.905,251.110,-71.342,-178.474,9.948,149.562
C01391=1117.900,251.359,-71.370,-178.471,9.950,149.562
C01392=1117.897,251.607,-71.399,-178.467,9.954,149.562
C01393=1117.892,251.855,-71.428,-178.464,9.957,149.562
C01394=1117.888,252.103,-71.456,-178.462,9.958,149.561
C01395=1117.883,252.352,-71.484,-178.459,9.961,149.561
C01396=1117.880,252.600,-71.513,-178.456,9.964,149.561
C01397=1117.876,252.814,-71.537,-178.453,9.966,149.561
C01398=1117.872,253.026,-71.562,-178.452,9.967,149.561
C01399=1117.869,253.239,-71.587,-178.449,9.969,149.561
C01400=1117.864,253.453,-71.611,-178.448,9.971,149.561
C01401=1117.861,253.666,-71.636,-178.446,9.972,149.561
C01402=1117.857,253.879,-71.660,-178.444,9.974,149.561
C01403=1117.853,254.093,-71.685,-178.442,9.976,149.561
C01404=1117.850,254.305,-71.709,-178.440,9.978,149.561
C01405=1117.845,254.554,-71.738,-178.439,9.979,149.561
C01406=1117.842,254.802,-71.767,-178.437,9.982,149.561
C01407=1117.837,255.050,-71.795,-178.436,9.983,149.561
C01408=1117.833,255.298,-71.824,-178.434,9.985,149.561
C01409=1117.829,255.547,-71.853,-178.433,9.987,149.561
C01410=1117.824,255.795,-71.881,-178.432,9.988,149.561
C01411=1117.820,256.043,-71.910,-178.431,9.991,149.561
C01412=1117.816,256.292,-71.939,-178.428,9.993,149.561
C01413=1117.811,256.539,-71.968,-178.425,9.996,149.561
C01414=1117.807,256.788,-71.996,-178.422,9.999,149.561
C01415=1117.803,257.036,-72.025,-178.420,10.002,149.561
C01416=1117.799,257.285,-72.054,-178.417,10.004,149.561
C01417=1117.794,257.533,-72.082,-178.414,10.007,149.561
C01418=1117.790,257.781,-72.111,-178.411,10.010,149.561
C01419=1117.786,258.030,-72.140,-178.408,10.013,149.561
C01420=1117.782,258.279,-72.169,-178.405,10.015,149.560
C01421=1117.778,258.526,-72.198,-178.403,10.019,149.561
C01422=1117.773,258.775,-72.227,-178.400,10.021,149.560
C01423=1117.769,259.023,-72.256,-178.397,10.024,149.560
C01424=1117.765,259.271,-72.284,-178.394,10.027,149.560
C01425=1117.760,259.519,-72.313,-178.390,10.030,149.560
C01426=1117.756,259.768,-72.342,-178.387,10.033,149.560
C01427=1117.752,260.016,-72.372,-178.384,10.036,149.560
C01428=1117.747,260.264,-72.401,-178.382,10.039,149.560
C01429=1117.744,260.513,-72.429,-178.379,10.041,149.560
C01430=1117.739,260.761,-72.458,-178.376,10.044,149.560
C01431=1117.735,261.009,-72.488,-178.373,10.047,149.559
C01432=1117.730,261.258,-72.516,-178.369,10.050,149.559
C01433=1117.726,261.506,-72.546,-178.366,10.053,149.559
C01434=1117.723,261.754,-72.575,-178.363,10.056,149.559
C01435=1117.718,262.002,-72.604,-178.360,10.058,149.559
C01436=1117.713,262.250,-72.633,-178.357,10.061,149.559
C01437=1117.709,262.499,-72.662,-178.353,10.064,149.558
C01438=1117.705,262.747,-72.691,-178.350,10.067,149.558
C01439=1117.701,262.995,-72.721,-178.347,10.070,149.558
C01440=1117.697,263.244,-72.750,-178.344,10.072,149.558
C01441=1117.692,263.492,-72.779,-178.340,10.076,149.558
C01442=1117.688,263.740,-72.808,-178.337,10.078,149.558
C01443=1117.684,263.988,-72.837,-178.334,10.081,149.557
C01444=1117.680,264.236,-72.866,-178.330,10.084,149.557
C01445=1117.676,264.484,-72.896,-178.327,10.087,149.557
C01446=1117.671,264.733,-72.925,-178.324,10.090,149.557
C01447=1117.667,264.981,-72.955,-178.322,10.092,149.557
C01448=1117.663,265.229,-72.984,-178.319,10.094,149.557
C01449=1117.659,265.478,-73.013,-178.316,10.096,149.557
C01450=1117.654,265.726,-73.042,-178.314,10.099,149.557
C01451=1117.650,265.974,-73.072,-178.311,10.102,149.556
C01452=1117.645,266.222,-73.101,-178.308,10.104,149.556
C01453=1117.642,266.435,-73.127,-178.306,10.106,149.556
C01454=1117.639,266.648,-73.152,-178.304,10.108,149.556
C01455=1117.635,266.862,-73.177,-178.302,10.110,149.556
C01456=1117.631,267.074,-73.203,-178.299,10.113,149.556
C01457=1117.628,267.287,-73.228,-178.297,10.115,149.556
C01458=1117.624,267.501,-73.253,-178.294,10.117,149.556
C01459=1117.620,267.714,-73.278,-178.292,10.119,149.556
C01460=1117.617,267.926,-73.304,-178.290,10.121,149.556
C01461=1117.612,268.175,-73.333,-178.287,10.124,149.555
C01462=1117.608,268.423,-73.363,-178.284,10.126,149.555
C01463=1117.604,268.671,-73.392,-178.281,10.128,149.555
C01464=1117.600,268.919,-73.422,-178.278,10.131,149.555
C01465=1117.595,269.168,-73.452,-178.276,10.134,149.555
C01466=1117.591,269.416,-73.482,-178.273,10.137,149.555
C01467=1117.587,269.664,-73.511,-178.270,10.139,149.555
C01468=1117.583,269.912,-73.541,-178.267,10.141,149.555
C01469=1117.579,270.160,-73.570,-178.264,10.144,149.555
C01470=1117.574,270.409,-73.600,-178.261,10.147,149.554
C01471=1117.570,270.657,-73.629,-178.259,10.149,149.554
C01472=1117.566,270.905,-73.659,-178.256,10.152,149.554
C01473=1117.561,271.153,-73.689,-178.253,10.154,149.554
C01474=1117.557,271.401,-73.719,-178.250,10.157,149.554
C01475=1117.553,271.650,-73.748,-178.247,10.160,149.554
C01476=1117.549,271.897,-73.778,-178.244,10.163,149.554
C01477=1117.545,272.146,-73.808,-178.242,10.165,149.554
C01478=1117.540,272.394,-73.838,-178.239,10.167,149.554
C01479=1117.536,272.642,-73.868,-178.236,10.170,149.554
C01480=1117.532,272.890,-73.898,-178.233,10.173,149.553
C01481=1117.528,273.138,-73.927,-178.230,10.176,149.553
C01482=1117.525,273.387,-73.958,-178.227,10.178,149.553
C01483=1117.520,273.635,-73.988,-178.225,10.181,149.553
C01484=1117.515,273.884,-74.017,-178.221,10.184,149.553
C01485=1117.512,274.131,-74.047,-178.218,10.186,149.553
C01486=1117.507,274.379,-74.077,-178.215,10.189,149.553
C01487=1117.503,274.627,-74.107,-178.213,10.191,149.553
C01488=1117.499,274.876,-74.137,-178.210,10.194,149.552
C01489=1117.495,275.123,-74.167,-178.207,10.197,149.552
C01490=1117.490,275.372,-74.197,-178.204,10.199,149.552
C01491=1117.486,275.621,-74.227,-178.201,10.202,149.552
C01492=1117.482,275.869,-74.257,-178.198,10.205,149.552
C01493=1117.478,276.117,-74.288,-178.195,10.207,149.552
C01494=1117.474,276.365,-74.317,-178.192,10.210,149.552
C01495=1117.470,276.612,-74.348,-178.189,10.212,149.551
C01496=1117.465,276.861,-74.378,-178.186,10.215,149.551
C01497=1117.461,277.109,-74.408,-178.183,10.218,149.551
C01498=1117.457,277.358,-74.438,-178.180,10.221,149.551
C01499=1117.453,277.606,-74.468,-178.177,10.223,149.551
C01500=1117.448,277.854,-74.498,-178.174,10.226,149.551
C01501=1117.445,278.101,-74.528,-178.171,10.229,149.551
C01502=1117.440,278.349,-74.559,-178.167,10.231,149.550
C01503=1117.436,278.598,-74.589,-178.164,10.234,149.550
C01504=1117.432,278.846,-74.619,-178.160,10.237,149.550
C01505=1117.428,279.094,-74.649,-178.157,10.240,149.550
C01506=1117.423,279.343,-74.680,-178.155,10.243,149.550
C01507=1117.419,279.590,-74.710,-178.151,10.245,149.549
C01508=1117.415,279.839,-74.741,-178.148,10.248,149.549
C01509=1117.412,280.052,-74.767,-178.146,10.250,149.549
C01510=1117.408,280.264,-74.792,-178.143,10.252,149.549
C01511=1117.404,280.477,-74.819,-178.140,10.254,149.549
C01512=1117.401,280.690,-74.845,-178.137,10.257,149.549
C01513=1117.397,280.903,-74.871,-178.135,10.259,149.548
C01514=1117.394,281.116,-74.897,-178.132,10.261,149.548
C01515=1117.390,281.328,-74.923,-178.129,10.264,149.548
C01516=1117.386,281.541,-74.949,-178.126,10.266,149.548
C01517=1117.382,281.789,-74.980,-178.123,10.268,149.548
C01518=1117.378,282.038,-75.010,-178.120,10.271,149.548
C01519=1117.374,282.286,-75.040,-178.117,10.274,149.547
C01520=1117.370,282.534,-75.071,-178.114,10.276,149.547
C01521=1117.365,282.782,-75.102,-178.111,10.278,149.547
C01522=1117.362,283.030,-75.132,-178.108,10.281,149.547
C01523=1117.357,283.278,-75.163,-178.105,10.284,149.547
C01524=1117.353,283.526,-75.193,-178.102,10.286,149.547
C01525=1117.349,283.775,-75.224,-178.099,10.289,149.547
C01526=1117.345,284.023,-75.255,-178.096,10.291,149.546
C01527=1117.341,284.270,-75.285,-178.093,10.294,149.546
C01528=1117.337,284.519,-75.316,-178.089,10.296,149.546
C01529=1117.332,284.767,-75.347,-178.087,10.299,149.546
C01530=1117.328,285.014,-75.377,-178.084,10.301,149.546
C01531=1117.324,285.263,-75.408,-178.081,10.303,149.545
C01532=1117.320,285.511,-75.439,-178.078,10.306,149.545
C01533=1117.316,285.759,-75.469,-178.075,10.309,149.545
C01534=1117.312,286.007,-75.500,-178.072,10.311,149.545
C01535=1117.307,286.255,-75.531,-178.068,10.314,149.545
C01536=1117.303,286.503,-75.561,-178.065,10.317,149.545
C01537=1117.299,286.752,-75.593,-178.062,10.319,149.544
C01538=1117.295,287.000,-75.623,-178.059,10.322,149.544
C01539=1117.290,287.248,-75.654,-178.057,10.324,149.544
C01540=1117.287,287.495,-75.685,-178.053,10.326,149.544
C01541=1117.282,287.743,-75.716,-178.051,10.329,149.544
C01542=1117.278,287.992,-75.747,-178.047,10.331,149.543
C01543=1117.274,288.240,-75.778,-178.044,10.334,149.543
C01544=1117.270,288.488,-75.808,-178.041,10.337,149.543
C01545=1117.266,288.736,-75.840,-178.038,10.339,149.543
C01546=1117.262,288.984,-75.871,-178.035,10.342,149.543
C01547=1117.258,289.232,-75.902,-178.032,10.345,149.543
C01548=1117.253,289.480,-75.933,-178.029,10.347,149.543
C01549=1117.250,289.728,-75.964,-178.026,10.349,149.542
C01550=1117.245,289.976,-75.995,-178.023,10.352,149.542
C01551=1117.241,290.224,-76.025,-178.020,10.354,149.542
C01552=1117.237,290.472,-76.057,-178.017,10.357,149.542
C01553=1117.232,290.720,-76.088,-178.014,10.359,149.542
C01554=1117.228,290.968,-76.119,-178.011,10.362,149.541
C01555=1117.224,291.216,-76.151,-178.008,10.365,149.541
C01556=1117.221,291.464,-76.181,-178.004,10.367,149.541
C01557=1117.216,291.712,-76.212,-178.001,10.370,149.541
C01558=1117.212,291.960,-76.244,-177.999,10.372,149.541
C01559=1117.208,292.208,-76.275,-177.996,10.374,149.541
C01560=1117.204,292.456,-76.306,-177.992,10.377,149.540
C01561=1117.200,292.704,-76.337,-177.989,10.380,149.540
C01562=1117.196,292.952,-76.369,-177.986,10.382,149.540
C01563=1117.191,293.200,-76.400,-177.983,10.385,149.540
C01564=1117.188,293.448,-76.432,-177.980,10.387,149.540
C01565=1117.184,293.661,-76.457,-177.978,10.389,149.539
C01566=1117.181,293.873,-76.485,-177.975,10.391,149.539
C01567=1117.177,294.086,-76.511,-177.972,10.394,149.539
C01568=1117.173,294.299,-76.538,-177.970,10.396,149.539
C01569=1117.171,294.512,-76.565,-177.967,10.398,149.539
C01570=1117.167,294.725,-76.592,-177.964,10.400,149.539
C01571=1117.163,294.937,-76.619,-177.962,10.402,149.539
C01572=1117.159,295.150,-76.646,-177.959,10.405,149.538
C01573=1117.155,295.399,-76.677,-177.956,10.407,149.538
C01574=1117.151,295.646,-76.709,-177.953,10.409,149.538
C01575=1117.147,295.894,-76.741,-177.950,10.412,149.538
C01576=1117.143,296.142,-76.772,-177.947,10.414,149.538
C01577=1117.139,296.390,-76.803,-177.944,10.417,149.538
C01578=1117.135,296.638,-76.835,-177.941,10.420,149.537
C01579=1117.131,296.886,-76.866,-177.938,10.422,149.537
C01580=1117.127,297.134,-76.898,-177.934,10.425,149.537
C01581=1117.123,297.381,-76.929,-177.931,10.428,149.537
C01582=1117.118,297.630,-76.960,-177.928,10.430,149.537
C01583=1117.114,297.878,-76.993,-177.926,10.432,149.537
C01584=1117.110,298.126,-77.024,-177.923,10.435,149.536
C01585=1117.106,298.374,-77.056,-177.919,10.437,149.536
C01586=1117.102,298.621,-77.088,-177.917,10.440,149.536
C01587=1117.098,298.870,-77.119,-177.913,10.442,149.536
C01588=1117.094,299.118,-77.151,-177.910,10.445,149.536
C01589=1117.090,299.365,-77.182,-177.907,10.448,149.535
C01590=1117.085,299.613,-77.215,-177.904,10.450,149.535
C01591=1117.082,299.861,-77.246,-177.901,10.453,149.535
C01592=1117.077,300.109,-77.278,-177.898,10.456,149.535
C01593=1117.073,300.357,-77.309,-177.895,10.457,149.535
C01594=1117.070,300.606,-77.341,-177.892,10.460,149.535
C01595=1117.064,300.853,-77.373,-177.889,10.462,149.534
C01596=1117.061,301.101,-77.405,-177.886,10.465,149.534
C01597=1117.057,301.349,-77.437,-177.883,10.468,149.534
C01598=1117.053,301.597,-77.468,-177.880,10.470,149.534
C01599=1117.048,301.845,-77.501,-177.876,10.473,149.534
C01600=1117.045,302.093,-77.532,-177.873,10.476,149.534
C01601=1117.040,302.340,-77.564,-177.870,10.478,149.533
C01602=1117.036,302.589,-77.596,-177.867,10.480,149.533
C01603=1117.032,302.837,-77.628,-177.864,10.482,149.533
C01604=1117.028,303.085,-77.660,-177.861,10.485,149.533
C01605=1117.023,303.332,-77.692,-177.858,10.488,149.533
C01606=1117.020,303.580,-77.724,-177.855,10.490,149.532
C01607=1117.016,303.828,-77.756,-177.852,10.493,149.532
C01608=1117.011,304.076,-77.788,-177.848,10.495,149.532
C01609=1117.007,304.324,-77.820,-177.846,10.498,149.532
C01610=1117.004,304.572,-77.852,-177.842,10.500,149.532
C01611=1116.999,304.820,-77.885,-177.839,10.503,149.532
C01612=1116.995,305.067,-77.916,-177.836,10.506,149.531
C01613=1116.991,305.315,-77.948,-177.833,10.508,149.531
C01614=1116.987,305.564,-77.980,-177.830,10.510,149.531
C01615=1116.983,305.812,-78.012,-177.827,10.513,149.531
C01616=1116.979,306.060,-78.045,-177.824,10.515,149.531
C01617=1116.975,306.307,-78.077,-177.821,10.518,149.531
C01618=1116.970,306.555,-78.109,-177.818,10.521,149.530
C01619=1116.967,306.803,-78.141,-177.815,10.523,149.530
C01620=1116.963,307.051,-78.173,-177.812,10.526,149.530
C01621=1116.959,307.263,-78.202,-177.809,10.528,149.530
C01622=1116.955,307.476,-78.229,-177.806,10.530,149.530
C01623=1116.952,307.689,-78.256,-177.804,10.532,149.530
C01624=1116.949,307.901,-78.284,-177.801,10.534,149.529
C01625=1116.946,308.114,-78.312,-177.798,10.537,149.529
C01626=1116.942,308.327,-78.339,-177.796,10.539,149.529
C01627=1116.938,308.539,-78.368,-177.793,10.541,149.529
C01628=1116.935,308.752,-78.395,-177.790,10.543,149.529
C01629=1116.931,309.000,-78.427,-177.787,10.546,149.529
C01630=1116.926,309.247,-78.460,-177.784,10.548,149.528
C01631=1116.923,309.495,-78.492,-177.782,10.550,149.528
C01632=1116.918,309.743,-78.525,-177.778,10.553,149.528
C01633=1116.915,309.991,-78.557,-177.775,10.555,149.528
C01634=1116.910,310.239,-78.589,-177.772,10.558,149.528
C01635=1116.906,310.487,-78.622,-177.769,10.560,149.527
C01636=1116.902,310.735,-78.654,-177.766,10.563,149.527
C01637=1116.898,310.983,-78.687,-177.762,10.566,149.527
C01638=1116.894,311.230,-78.719,-177.759,10.568,149.527
C01639=1116.890,311.478,-78.752,-177.756,10.571,149.527
C01640=1116.885,311.726,-78.784,-177.753,10.574,149.527
C01641=1116.882,311.973,-78.817,-177.750,10.576,149.526
C01642=1116.878,312.222,-78.849,-177.747,10.578,149.526
C01643=1116.874,312.469,-78.882,-177.744,10.580,149.526
C01644=1116.870,312.717,-78.915,-177.741,10.583,149.526
C01645=1116.866,312.965,-78.947,-177.738,10.586,149.526
C01646=1116.862,313.213,-78.980,-177.735,10.588,149.525
C01647=1116.858,313.461,-79.012,-177.732,10.591,149.525
C01648=1116.854,313.709,-79.046,-177.728,10.593,149.525
C01649=1116.850,313.956,-79.078,-177.725,10.596,149.525
C01650=1116.846,314.205,-79.111,-177.722,10.598,149.525
C01651=1116.842,314.452,-79.144,-177.719,10.601,149.525
C01652=1116.838,314.700,-79.176,-177.716,10.604,149.525
C01653=1116.834,314.948,-79.209,-177.713,10.605,149.524
C01654=1116.830,315.196,-79.242,-177.710,10.608,149.524
C01655=1116.825,315.444,-79.275,-177.707,10.611,149.524
C01656=1116.822,315.691,-79.308,-177.704,10.613,149.524
C01657=1116.818,315.939,-79.340,-177.701,10.616,149.524
C01658=1116.813,316.187,-79.373,-177.697,10.618,149.523
C01659=1116.809,316.435,-79.406,-177.694,10.621,149.523
C01660=1116.806,316.682,-79.439,-177.691,10.623,149.523
C01661=1116.802,316.930,-79.472,-177.688,10.626,149.523
C01662=1116.797,317.178,-79.505,-177.685,10.629,149.523
C01663=1116.793,317.426,-79.538,-177.682,10.631,149.522
C01664=1116.790,317.673,-79.570,-177.679,10.633,149.522
C01665=1116.786,317.921,-79.603,-177.676,10.635,149.522
C01666=1116.782,318.169,-79.637,-177.673,10.638,149.522
C01667=1116.777,318.417,-79.670,-177.670,10.641,149.522
C01668=1116.773,318.664,-79.703,-177.666,10.643,149.522
C01669=1116.769,318.912,-79.736,-177.663,10.646,149.521
C01670=1116.766,319.159,-79.769,-177.660,10.648,149.521
C01671=1116.762,319.407,-79.802,-177.657,10.651,149.521
C01672=1116.757,319.655,-79.835,-177.654,10.654,149.521
C01673=1116.754,319.903,-79.868,-177.650,10.656,149.521
C01674=1116.750,320.151,-79.902,-177.647,10.658,149.520
C01675=1116.746,320.399,-79.935,-177.644,10.661,149.520
C01676=1116.741,320.647,-79.968,-177.642,10.663,149.520
C01677=1116.739,320.859,-79.996,-177.639,10.666,149.520
C01678=1116.735,321.071,-80.025,-177.636,10.667,149.520
C01679=1116.732,321.284,-80.053,-177.633,10.670,149.520
C01680=1116.728,321.496,-80.082,-177.630,10.672,149.519
C01681=1116.725,321.709,-80.110,-177.628,10.674,149.519
C01682=1116.721,321.921,-80.139,-177.625,10.677,149.519
C01683=1116.717,322.134,-80.167,-177.622,10.678,149.519
C01684=1116.714,322.346,-80.196,-177.620,10.680,149.519
C01685=1116.710,322.594,-80.229,-177.617,10.683,149.519
C01686=1116.706,322.842,-80.262,-177.614,10.685,149.518
C01687=1116.702,323.089,-80.295,-177.611,10.688,149.518
C01688=1116.699,323.337,-80.329,-177.607,10.690,149.518
C01689=1116.695,323.585,-80.362,-177.604,10.693,149.518
C01690=1116.691,323.833,-80.396,-177.601,10.696,149.518
C01691=1116.686,324.080,-80.429,-177.598,10.698,149.517
C01692=1116.682,324.328,-80.462,-177.595,10.701,149.517
C01693=1116.678,324.575,-80.496,-177.591,10.703,149.517
C01694=1116.675,324.824,-80.529,-177.589,10.705,149.517
C01695=1116.671,325.071,-80.562,-177.586,10.708,149.517
C01696=1116.667,325.318,-80.596,-177.582,10.710,149.517
C01697=1116.662,325.567,-80.630,-177.579,10.713,149.516
C01698=1116.658,325.814,-80.663,-177.576,10.715,149.516
C01699=1116.655,326.062,-80.697,-177.573,10.718,149.516
C01700=1116.651,326.310,-80.731,-177.570,10.720,149.516
C01701=1116.646,326.558,-80.764,-177.567,10.723,149.516
C01702=1116.643,326.805,-80.798,-177.563,10.725,149.515
C01703=1116.639,327.053,-80.831,-177.560,10.728,149.515
C01704=1116.635,327.300,-80.865,-177.557,10.731,149.515
C01705=1116.630,327.548,-80.899,-177.554,10.733,149.515
C01706=1116.626,327.796,-80.932,-177.551,10.735,149.515
C01707=1116.623,328.044,-80.966,-177.548,10.738,149.515
C01708=1116.619,328.291,-80.999,-177.545,10.740,149.514
C01709=1116.615,328.539,-81.033,-177.541,10.743,149.514
C01710=1116.610,328.787,-81.067,-177.539,10.745,149.514
C01711=1116.607,329.034,-81.101,-177.535,10.748,149.514
C01712=1116.603,329.282,-81.134,-177.532,10.750,149.514
C01713=1116.599,329.529,-81.168,-177.529,10.753,149.513
C01714=1116.595,329.778,-81.202,-177.526,10.755,149.513
C01715=1116.591,330.025,-81.236,-177.522,10.758,149.513
C01716=1116.587,330.272,-81.270,-177.519,10.760,149.513
C01717=1116.583,330.521,-81.304,-177.516,10.763,149.513
C01718=1116.579,330.768,-81.338,-177.513,10.765,149.512
C01719=1116.575,331.016,-81.371,-177.510,10.767,149.512
C01720=1116.572,331.264,-81.405,-177.507,10.770,149.512
C01721=1116.568,331.511,-81.439,-177.504,10.772,149.512
C01722=1116.563,331.759,-81.473,-177.501,10.775,149.512
C01723=1116.560,332.007,-81.507,-177.497,10.777,149.511
C01724=1116.556,332.254,-81.541,-177.494,10.780,149.511
C01725=1116.551,332.502,-81.575,-177.491,10.783,149.511
C01726=1116.548,332.750,-81.609,-177.488,10.785,149.511
C01727=1116.544,332.997,-81.643,-177.485,10.788,149.511
C01728=1116.539,333.244,-81.677,-177.481,10.790,149.511
C01729=1116.536,333.493,-81.711,-177.478,10.793,149.510
C01730=1116.531,333.740,-81.745,-177.475,10.794,149.510
C01731=1116.528,333.988,-81.780,-177.473,10.797,149.510
C01732=1116.524,334.235,-81.814,-177.469,10.800,149.510
C01733=1116.521,334.447,-81.843,-177.466,10.802,149.510
C01734=1116.517,334.660,-81.872,-177.464,10.804,149.509
C01735=1116.514,334.872,-81.901,-177.461,10.806,149.509
C01736=1116.510,335.084,-81.931,-177.458,10.809,149.509
C01737=1116.507,335.297,-81.960,-177.455,10.810,149.509
C01738=1116.504,335.509,-81.989,-177.453,10.812,149.509
C01739=1116.500,335.721,-82.019,-177.450,10.815,149.509
C01740=1116.497,335.933,-82.049,-177.447,10.817,149.508
C01741=1116.493,336.181,-82.082,-177.444,10.819,149.508
C01742=1116.489,336.429,-82.117,-177.441,10.822,149.508
C01743=1116.485,336.676,-82.150,-177.438,10.824,149.508
C01744=1116.481,336.924,-82.185,-177.435,10.827,149.508
C01745=1116.477,337.172,-82.219,-177.431,10.829,149.507
C01746=1116.473,337.419,-82.254,-177.428,10.832,149.507
C01747=1116.470,337.667,-82.288,-177.425,10.835,149.507
C01748=1116.465,337.914,-82.322,-177.422,10.837,149.507
C01749=1116.461,338.162,-82.357,-177.419,10.839,149.507
C01750=1116.457,338.409,-82.391,-177.416,10.841,149.506
C01751=1116.453,338.658,-82.426,-177.413,10.844,149.506
C01752=1116.450,338.904,-82.460,-177.409,10.846,149.506
C01753=1116.446,339.152,-82.495,-177.406,10.849,149.506
C01754=1116.442,339.399,-82.529,-177.403,10.851,149.506
C01755=1116.438,339.647,-82.564,-177.400,10.854,149.506
C01756=1116.433,339.895,-82.598,-177.397,10.856,149.505
C01757=1116.430,340.143,-82.633,-177.393,10.859,149.505
C01758=1116.426,340.390,-82.667,-177.390,10.861,149.505
C01759=1116.422,340.638,-82.702,-177.387,10.864,149.505
C01760=1116.418,340.885,-82.737,-177.384,10.867,149.505
C01761=1116.414,341.133,-82.771,-177.381,10.868,149.504
C01762=1116.410,341.380,-82.806,-177.378,10.871,149.504
C01763=1116.406,341.628,-82.840,-177.374,10.873,149.504
C01764=1116.402,341.875,-82.875,-177.371,10.876,149.504
C01765=1116.398,342.123,-82.910,-177.368,10.878,149.504
C01766=1116.395,342.371,-82.944,-177.365,10.881,149.503
C01767=1116.390,342.618,-82.979,-177.362,10.883,149.503
C01768=1116.387,342.866,-83.014,-177.358,10.886,149.503
C01769=1116.382,343.113,-83.049,-177.355,10.889,149.503
C01770=1116.379,343.361,-83.083,-177.352,10.891,149.503
C01771=1116.375,343.608,-83.119,-177.349,10.894,149.502
C01772=1116.371,343.856,-83.153,-177.345,10.896,149.502
C01773=1116.367,344.104,-83.188,-177.343,10.898,149.502
C01774=1116.363,344.350,-83.222,-177.339,10.900,149.502
C01775=1116.359,344.599,-83.257,-177.336,10.903,149.502
C01776=1116.355,344.846,-83.293,-177.333,10.905,149.501
C01777=1116.351,345.093,-83.327,-177.330,10.908,149.501
C01778=1116.348,345.341,-83.362,-177.326,10.910,149.501
C01779=1116.343,345.588,-83.397,-177.323,10.913,149.501
C01780=1116.340,345.836,-83.432,-177.320,10.916,149.501
C01781=1116.336,346.084,-83.467,-177.317,10.918,149.500
C01782=1116.332,346.331,-83.502,-177.314,10.920,149.500
C01783=1116.328,346.579,-83.537,-177.310,10.923,149.500
C01784=1116.325,346.826,-83.572,-177.307,10.925,149.500
C01785=1116.320,347.073,-83.607,-177.304,10.928,149.500
C01786=1116.316,347.321,-83.642,-177.301,10.930,149.499
C01787=1116.312,347.569,-83.677,-177.298,10.932,149.499
C01788=1116.308,347.816,-83.712,-177.295,10.935,149.499
C01789=1116.305,348.028,-83.742,-177.291,10.937,149.499
C01790=1116.302,348.241,-83.773,-177.289,10.939,149.499
C01791=1116.299,348.453,-83.803,-177.287,10.941,149.498
C01792=1116.295,348.665,-83.832,-177.284,10.944,149.498
C01793=1116.292,348.877,-83.863,-177.281,10.945,149.498
C01794=1116.289,349.089,-83.893,-177.278,10.947,149.498
C01795=1116.285,349.301,-83.924,-177.275,10.950,149.498
C01796=1116.282,349.513,-83.953,-177.273,10.952,149.498
C01797=1116.278,349.761,-83.989,-177.269,10.954,149.497
C01798=1116.274,350.008,-84.024,-177.266,10.956,149.497
C01799=1116.270,350.256,-84.059,-177.262,10.960,149.497
C01800=1116.266,350.503,-84.094,-177.259,10.962,149.497
C01801=1116.263,350.751,-84.130,-177.255,10.965,149.496
C01802=1116.258,350.998,-84.165,-177.252,10.967,149.496
C01803=1116.254,351.246,-84.200,-177.249,10.970,149.496
C01804=1116.251,351.493,-84.235,-177.246,10.972,149.496
C01805=1116.247,351.741,-84.271,-177.242,10.974,149.496
C01806=1116.243,351.988,-84.307,-177.239,10.977,149.495
C01807=1116.239,352.235,-84.342,-177.235,10.979,149.495
C01808=1116.235,352.483,-84.377,-177.231,10.982,149.495
C01809=1116.232,352.730,-84.413,-177.228,10.985,149.495
C01810=1116.228,352.978,-84.448,-177.225,10.987,149.494
C01811=1116.224,353.226,-84.483,-177.221,10.990,149.494
C01812=1116.220,353.473,-84.518,-177.218,10.992,149.494
C01813=1116.216,353.720,-84.554,-177.215,10.995,149.494
C01814=1116.212,353.968,-84.589,-177.211,10.997,149.493
C01815=1116.209,354.215,-84.625,-177.208,10.999,149.493
C01816=1116.204,354.463,-84.661,-177.204,11.002,149.493
C01817=1116.201,354.710,-84.697,-177.201,11.004,149.493
C01818=1116.197,354.957,-84.732,-177.198,11.007,149.492
C01819=1116.193,355.205,-84.767,-177.194,11.009,149.492
C01820=1116.189,355.452,-84.803,-177.191,11.012,149.492
C01821=1116.186,355.700,-84.839,-177.187,11.014,149.491
C01822=1116.182,355.947,-84.875,-177.184,11.016,149.491
C01823=1116.178,356.194,-84.911,-177.181,11.019,149.491
